LIN {X 0,Y 574.364,Z 450.837,A -85,B 0,C 180,E1 -2266.254,E2 -2266.254} C_VEL
LIN {X 0,Y 574.549,Z 436.626,A -85,B 0,C 180,E1 -2266.797,E2 -2266.797} C_VEL
LIN {X 0,Y 574.69,Z 422.126,A -85,B 0,C 180,E1 -2267.209,E2 -2267.209} C_VEL
LIN {X 0,Y 574.753,Z 406.706,A -85,B 0,C 180,E1 -2267.502,E2 -2267.502} C_VEL
LIN {X 0,Y 575.14,Z 251.823,A -85,B 0,C 180,E1 -2269.493,E2 -2269.493} C_VEL
LIN {X 0,Y 574.003,Z 245.811,A -85,B 0,C 180,E1 -2269.623,E2 -2269.623} C_VEL
LIN {X 0,Y 574.349,Z 220.396,A -85,B 0,C 180,E1 -2272.671,E2 -2272.671} C_VEL
LIN {X 0,Y 574.581,Z 198.331,A -85,B 0,C 180,E1 -2275.347,E2 -2275.347} C_VEL
LIN {X 0,Y 574.295,Z 195.164,A -85,B 0,C 180,E1 -2275.749,E2 -2275.749} C_VEL
LIN {X 0,Y 573.262,Z 190.706,A -85,B 0,C 180,E1 -2276.38,E2 -2276.38} C_VEL
LIN {X 0,Y 573.262,Z 190.698,A -85,B 0,C 180,E1 -2279.365,E2 -2279.365} C_VEL
LIN {X 0,Y 573.247,Z 190.706,A -85,B 0,C 180,E1 -2282.227,E2 -2282.227} C_VEL
LIN {X 0,Y 573.235,Z 190.701,A -85,B 0,C 180,E1 -2284.771,E2 -2284.771} C_VEL
LIN {X 0,Y 573.249,Z 190.698,A -85,B 0,C 180,E1 -2287.165,E2 -2287.165} C_VEL
LIN {X 0,Y 573.243,Z 190.702,A -85,B 0,C 180,E1 -2289.606,E2 -2289.606} C_VEL
LIN {X 0,Y 573.237,Z 190.701,A -85,B 0,C 180,E1 -2292.641,E2 -2292.641} C_VEL
LIN {X 0,Y 573.229,Z 190.705,A -85,B 0,C 180,E1 -2295.666,E2 -2295.666} C_VEL
LIN {X 0,Y 573.239,Z 190.7,A -85,B 0,C 180,E1 -2298.544,E2 -2298.544} C_VEL
LIN {X 0,Y 573.243,Z 190.7,A -85,B 0,C 180,E1 -2301.299,E2 -2301.299} C_VEL
LIN {X 0,Y 573.257,Z 190.704,A -85,B 0,C 180,E1 -2304.011,E2 -2304.011} C_VEL
LIN {X 0,Y 573.277,Z 190.695,A -85,B 0,C 180,E1 -2306.518,E2 -2306.518} C_VEL
LIN {X 0,Y 573.236,Z 190.7,A -85,B 0,C 180,E1 -2309.115,E2 -2309.115} C_VEL
LIN {X 0,Y 573.256,Z 190.703,A -85,B 0,C 180,E1 -2311.968,E2 -2311.968} C_VEL
LIN {X 0,Y 573.245,Z 190.699,A -85,B 0,C 180,E1 -2314.59,E2 -2314.59} C_VEL
LIN {X 0,Y 573.231,Z 190.707,A -85,B 0,C 180,E1 -2317.662,E2 -2317.662} C_VEL
LIN {X 0,Y 573.248,Z 190.703,A -85,B 0,C 180,E1 -2319.923,E2 -2319.923} C_VEL
LIN {X 0,Y 573.254,Z 190.699,A -85,B 0,C 180,E1 -2322.988,E2 -2322.988} C_VEL
LIN {X 0,Y 573.264,Z 190.702,A -85,B 0,C 180,E1 -2325.807,E2 -2325.807} C_VEL
LIN {X 0,Y 573.273,Z 190.695,A -85,B 0,C 180,E1 -2328.734,E2 -2328.734} C_VEL
LIN {X 0,Y 573.298,Z 190.701,A -85,B 0,C 180,E1 -2331.541,E2 -2331.541} C_VEL
LIN {X 0,Y 573.285,Z 190.693,A -85,B 0,C 180,E1 -2334.372,E2 -2334.372} C_VEL
LIN {X 0,Y 573.298,Z 190.695,A -85,B 0,C 180,E1 -2337.892,E2 -2337.892} C_VEL
LIN {X 0,Y 573.329,Z 190.688,A -85,B 0,C 180,E1 -2340.702,E2 -2340.702} C_VEL
LIN {X 0,Y 573.233,Z 190.706,A -85,B 0,C 180,E1 -2343.515,E2 -2343.515} C_VEL
LIN {X 0,Y 573.287,Z 190.698,A -85,B 0,C 180,E1 -2345.628,E2 -2345.628} C_VEL
LIN {X 0,Y 573.299,Z 190.691,A -85,B 0,C 180,E1 -2348.459,E2 -2348.459} C_VEL
LIN {X 0,Y 573.29,Z 190.701,A -85,B 0,C 180,E1 -2351.312,E2 -2351.312} C_VEL
LIN {X 0,Y 573.272,Z 190.696,A -85,B 0,C 180,E1 -2354.425,E2 -2354.425} C_VEL
LIN {X 0,Y 573.251,Z 190.707,A -85,B 0,C 180,E1 -2357.112,E2 -2357.112} C_VEL
LIN {X 0,Y 573.246,Z 190.698,A -85,B 0,C 180,E1 -2360.077,E2 -2360.077} C_VEL
LIN {X 0,Y 573.225,Z 190.71,A -85,B 0,C 180,E1 -2363.1,E2 -2363.1} C_VEL
LIN {X 0,Y 573.243,Z 190.699,A -85,B 0,C 180,E1 -2364.399,E2 -2364.399} C_VEL
LIN {X 0,Y 572.617,Z 190.785,A -85,B 0,C 180,E1 -2364.985,E2 -2364.985} C_VEL
LIN {X 0,Y 569.775,Z 191.14,A -85,B 0,C 180,E1 -2365.937,E2 -2365.937} C_VEL
LIN {X 0,Y 567.345,Z 191.442,A -85,B 0,C 180,E1 -2366.702,E2 -2366.702} C_VEL
LIN {X 0,Y 566.294,Z 191.569,A -85,B 0,C 180,E1 -2367.294,E2 -2367.294} C_VEL
LIN {X 0,Y 566.206,Z 191.578,A -85,B 0,C 180,E1 -2367.494,E2 -2367.494} C_VEL
LIN {X 0,Y 566.219,Z 191.574,A -85,B 0,C 180,E1 -2369.768,E2 -2369.768} C_VEL
LIN {X 0,Y 566.2,Z 191.579,A -85,B 0,C 180,E1 -2372.431,E2 -2372.431} C_VEL
LIN {X 0,Y 566.208,Z 191.584,A -85,B 0,C 180,E1 -2374.995,E2 -2374.995} C_VEL
LIN {X 0,Y 566.191,Z 191.579,A -85,B 0,C 180,E1 -2377.461,E2 -2377.461} C_VEL
LIN {X 0,Y 566.222,Z 191.574,A -85,B 0,C 180,E1 -2380.198,E2 -2380.198} C_VEL
LIN {X 0,Y 566.196,Z 191.582,A -85,B 0,C 180,E1 -2383.055,E2 -2383.055} C_VEL
LIN {X 0,Y 566.198,Z 191.577,A -85,B 0,C 180,E1 -2386.049,E2 -2386.049} C_VEL
LIN {X 0,Y 566.207,Z 191.584,A -85,B 0,C 180,E1 -2388.864,E2 -2388.864} C_VEL
LIN {X 0,Y 566.184,Z 191.578,A -85,B 0,C 180,E1 -2391.638,E2 -2391.638} C_VEL
LIN {X 0,Y 566.16,Z 191.586,A -85,B 0,C 180,E1 -2394.309,E2 -2394.309} C_VEL
LIN {X 0,Y 566.228,Z 191.579,A -85,B 0,C 180,E1 -2396.899,E2 -2396.899} C_VEL
LIN {X 0,Y 566.182,Z 191.58,A -85,B 0,C 180,E1 -2399.408,E2 -2399.408} C_VEL
LIN {X 0,Y 566.211,Z 191.578,A -85,B 0,C 180,E1 -2401.858,E2 -2401.858} C_VEL
LIN {X 0,Y 566.214,Z 191.582,A -85,B 0,C 180,E1 -2404.252,E2 -2404.252} C_VEL
LIN {X 0,Y 566.209,Z 191.685,A -85,B 0,C 180,E1 -2406.549,E2 -2406.549} C_VEL
LIN {X 0,Y 567.22,Z 197.326,A -85,B 0,C 180,E1 -2407.413,E2 -2407.413} C_VEL
LIN {X 0,Y 566.915,Z 216.903,A -85,B 0,C 180,E1 -2410.188,E2 -2410.188} C_VEL
LIN {X 0,Y 568.489,Z 225.078,A -85,B 0,C 180,E1 -2410.358,E2 -2410.358} C_VEL
LIN {X 0,Y 567.967,Z 382.291,A -85,B 0,C 180,E1 -2412.415,E2 -2412.415} C_VEL
LIN {X 0,Y 567.819,Z 397.78,A -85,B 0,C 180,E1 -2412.766,E2 -2412.766} C_VEL
LIN {X 0,Y 567.62,Z 413.086,A -85,B 0,C 180,E1 -2413.27,E2 -2413.27} C_VEL
LIN {X 0,Y 567.399,Z 427.739,A -85,B 0,C 180,E1 -2413.911,E2 -2413.911} C_VEL
LIN {X 0,Y 567.156,Z 441.053,A -85,B 0,C 180,E1 -2414.641,E2 -2414.641} C_VEL
LIN {X 0,Y 566.917,Z 453.985,A -85,B 0,C 180,E1 -2415.508,E2 -2415.508} C_VEL
LIN {X 0,Y 566.653,Z 466.893,A -85,B 0,C 180,E1 -2416.553,E2 -2416.553} C_VEL
LIN {X 0,Y 566.462,Z 478.088,A -85,B 0,C 180,E1 -2417.642,E2 -2417.642} C_VEL
LIN {X 0,Y 566.263,Z 488.18,A -85,B 0,C 180,E1 -2418.81,E2 -2418.81} C_VEL
LIN {X 0,Y 566.133,Z 498.005,A -85,B 0,C 180,E1 -2420.172,E2 -2420.172} C_VEL
LIN {X 0,Y 566.063,Z 505.495,A -85,B 0,C 180,E1 -2421.432,E2 -2421.432} C_VEL
LIN {X 0,Y 565.975,Z 512.5,A -85,B 0,C 180,E1 -2422.867,E2 -2422.867} C_VEL
LIN {X 0,Y 565.982,Z 518.009,A -85,B 0,C 180,E1 -2424.299,E2 -2424.299} C_VEL
LIN {X 0,Y 565.913,Z 522.178,A -85,B 0,C 180,E1 -2425.727,E2 -2425.727} C_VEL
LIN {X 0,Y 565.872,Z 525.113,A -85,B 0,C 180,E1 -2427.152,E2 -2427.152} C_VEL
LIN {X 0,Y 565.842,Z 526.879,A -85,B 0,C 180,E1 -2428.577,E2 -2428.577} C_VEL
LIN {X 0,Y 565.837,Z 527.496,A -85,B 0,C 180,E1 -2430,E2 -2430} C_VEL
LIN {X 0,Y 565.844,Z 526.941,A -85,B 0,C 180,E1 -2431.423,E2 -2431.423} C_VEL
LIN {X 0,Y 565.874,Z 525.257,A -85,B 0,C 180,E1 -2432.847,E2 -2432.847} C_VEL
LIN {X 0,Y 565.913,Z 522.404,A -85,B 0,C 180,E1 -2434.273,E2 -2434.273} C_VEL
LIN {X 0,Y 565.975,Z 518.318,A -85,B 0,C 180,E1 -2435.701,E2 -2435.701} C_VEL
LIN {X 0,Y 565.975,Z 512.904,A -85,B 0,C 180,E1 -2437.133,E2 -2437.133} C_VEL
LIN {X 0,Y 566.061,Z 506.004,A -85,B 0,C 180,E1 -2438.568,E2 -2438.568} C_VEL
LIN {X 0,Y 566.177,Z 497.395,A -85,B 0,C 180,E1 -2440.008,E2 -2440.008} C_VEL
LIN {X 0,Y 566.25,Z 488.954,A -85,B 0,C 180,E1 -2441.183,E2 -2441.183} C_VEL
LIN {X 0,Y 566.436,Z 478.917,A -85,B 0,C 180,E1 -2442.358,E2 -2442.358} C_VEL
LIN {X 0,Y 566.668,Z 466.874,A -85,B 0,C 180,E1 -2443.538,E2 -2443.538} C_VEL
LIN {X 0,Y 566.878,Z 455.249,A -85,B 0,C 180,E1 -2444.488,E2 -2444.488} C_VEL
LIN {X 0,Y 567.091,Z 442.476,A -85,B 0,C 180,E1 -2445.361,E2 -2445.361} C_VEL
LIN {X 0,Y 567.376,Z 429.466,A -85,B 0,C 180,E1 -2446.09,E2 -2446.09} C_VEL
LIN {X 0,Y 567.567,Z 415.275,A -85,B 0,C 180,E1 -2446.732,E2 -2446.732} C_VEL
LIN {X 0,Y 567.789,Z 400.729,A -85,B 0,C 180,E1 -2447.235,E2 -2447.235} C_VEL
LIN {X 0,Y 567.928,Z 385.332,A -85,B 0,C 180,E1 -2447.615,E2 -2447.615} C_VEL
LIN {X 0,Y 568.048,Z 363.9,A -85,B 0,C 180,E1 -2447.932,E2 -2447.932} C_VEL
LIN {X 0,Y 568.437,Z 224.034,A -85,B 0,C 180,E1 -2449.748,E2 -2449.748} C_VEL
LIN {X 0,Y 566.883,Z 216.905,A -85,B 0,C 180,E1 -2449.903,E2 -2449.903} C_VEL
LIN {X 0,Y 567.213,Z 199.31,A -85,B 0,C 180,E1 -2452.395,E2 -2452.395} C_VEL
LIN {X 0,Y 567.005,Z 195.381,A -85,B 0,C 180,E1 -2452.971,E2 -2452.971} C_VEL
LIN {X 0,Y 566.191,Z 191.587,A -85,B 0,C 180,E1 -2453.573,E2 -2453.573} C_VEL
LIN {X 0,Y 566.215,Z 191.583,A -85,B 0,C 180,E1 -2455.748,E2 -2455.748} C_VEL
LIN {X 0,Y 566.202,Z 191.579,A -85,B 0,C 180,E1 -2458.201,E2 -2458.201} C_VEL
LIN {X 0,Y 566.192,Z 191.582,A -85,B 0,C 180,E1 -2461.076,E2 -2461.076} C_VEL
LIN {X 0,Y 566.21,Z 191.581,A -85,B 0,C 180,E1 -2463.734,E2 -2463.734} C_VEL
LIN {X 0,Y 566.205,Z 191.576,A -85,B 0,C 180,E1 -2466.569,E2 -2466.569} C_VEL
LIN {X 0,Y 566.208,Z 191.58,A -85,B 0,C 180,E1 -2469.685,E2 -2469.685} C_VEL
LIN {X 0,Y 566.21,Z 191.576,A -85,B 0,C 180,E1 -2472.086,E2 -2472.086} C_VEL
LIN {X 0,Y 566.169,Z 191.586,A -85,B 0,C 180,E1 -2475.035,E2 -2475.035} C_VEL
LIN {X 0,Y 566.212,Z 191.573,A -85,B 0,C 180,E1 -2478.135,E2 -2478.135} C_VEL
LIN {X 0,Y 566.217,Z 191.577,A -85,B 0,C 180,E1 -2480.726,E2 -2480.726} C_VEL
LIN {X 0,Y 566.212,Z 191.576,A -85,B 0,C 180,E1 -2483.783,E2 -2483.783} C_VEL
LIN {X 0,Y 566.205,Z 191.576,A -85,B 0,C 180,E1 -2486.265,E2 -2486.265} C_VEL
LIN {X 0,Y 566.196,Z 191.58,A -85,B 0,C 180,E1 -2488.921,E2 -2488.921} C_VEL
LIN {X 0,Y 566.189,Z 191.586,A -85,B 0,C 180,E1 -2491.046,E2 -2491.046} C_VEL
LIN {X 0,Y 566.208,Z 191.578,A -85,B 0,C 180,E1 -2493.458,E2 -2493.458} C_VEL
LIN {X 0,Y 566.192,Z 191.578,A -85,B 0,C 180,E1 -2495.819,E2 -2495.819} C_VEL
LIN {X 0,Y 566.208,Z 191.584,A -85,B 0,C 180,E1 -2498.902,E2 -2498.902} C_VEL
LIN {X 0,Y 566.204,Z 191.581,A -85,B 0,C 180,E1 -2501.172,E2 -2501.172} C_VEL
LIN {X 0,Y 566.213,Z 191.577,A -85,B 0,C 180,E1 -2503.412,E2 -2503.412} C_VEL
LIN {X 0,Y 566.193,Z 191.578,A -85,B 0,C 180,E1 -2506.359,E2 -2506.359} C_VEL
LIN {X 0,Y 566.266,Z 191.575,A -85,B 0,C 180,E1 -2508.654,E2 -2508.654} C_VEL
LIN {X 0,Y 566.226,Z 191.574,A -85,B 0,C 180,E1 -2511.434,E2 -2511.434} C_VEL
LIN {X 0,Y 566.254,Z 191.572,A -85,B 0,C 180,E1 -2514.302,E2 -2514.302} C_VEL
LIN {X 0,Y 566.269,Z 191.568,A -85,B 0,C 180,E1 -2517.866,E2 -2517.866} C_VEL
LIN {X 0,Y 566.3,Z 191.573,A -85,B 0,C 180,E1 -2520.711,E2 -2520.711} C_VEL
LIN {X 0,Y 566.271,Z 191.573,A -85,B 0,C 180,E1 -2522.845,E2 -2522.845} C_VEL
LIN {X 0,Y 566.252,Z 191.57,A -85,B 0,C 180,E1 -2525.698,E2 -2525.698} C_VEL
LIN {X 0,Y 566.239,Z 191.58,A -85,B 0,C 180,E1 -2528.565,E2 -2528.565} C_VEL
LIN {X 0,Y 566.241,Z 191.571,A -85,B 0,C 180,E1 -2531.454,E2 -2531.454} C_VEL
LIN {X 0,Y 566.224,Z 191.583,A -85,B 0,C 180,E1 -2534.507,E2 -2534.507} C_VEL
LIN {X 0,Y 566.195,Z 191.576,A -85,B 0,C 180,E1 -2537.332,E2 -2537.332} C_VEL
LIN {X 0,Y 566.211,Z 191.585,A -85,B 0,C 180,E1 -2540.337,E2 -2540.337} C_VEL
LIN {X 0,Y 566.181,Z 191.579,A -85,B 0,C 180,E1 -2543.404,E2 -2543.404} C_VEL
LIN {X 0,Y 566.205,Z 191.577,A -85,B 0,C 180,E1 -2545.749,E2 -2545.749} C_VEL
LIN {X 0,Y 566.198,Z 191.586,A -85,B 0,C 180,E1 -2548.204,E2 -2548.204} C_VEL
LIN {X 0,Y 566.186,Z 191.582,A -85,B 0,C 180,E1 -2550.592,E2 -2550.592} C_VEL
LIN {X 0,Y 566.221,Z 191.573,A -85,B 0,C 180,E1 -2553.102,E2 -2553.102} C_VEL
LIN {X 0,Y 566.205,Z 191.579,A -85,B 0,C 180,E1 -2555.689,E2 -2555.689} C_VEL
LIN {X 0,Y 566.206,Z 191.578,A -85,B 0,C 180,E1 -2558.559,E2 -2558.559} C_VEL
LIN {X 0,Y 566.205,Z 191.573,A -85,B 0,C 180,E1 -2561.137,E2 -2561.137} C_VEL
LIN {X 0,Y 566.191,Z 191.587,A -85,B 0,C 180,E1 -2564.036,E2 -2564.036} C_VEL
LIN {X 0,Y 566.199,Z 191.577,A -85,B 0,C 180,E1 -2567.083,E2 -2567.083} C_VEL
LIN {X 0,Y 566.222,Z 191.581,A -85,B 0,C 180,E1 -2569.803,E2 -2569.803} C_VEL
LIN {X 0,Y 566.195,Z 191.577,A -85,B 0,C 180,E1 -2572.6,E2 -2572.6} C_VEL
LIN {X 0,Y 566.204,Z 191.577,A -85,B 0,C 180,E1 -2575.183,E2 -2575.183} C_VEL
LIN {X 0,Y 566.227,Z 191.582,A -85,B 0,C 180,E1 -2577.744,E2 -2577.744} C_VEL
LIN {X 0,Y 566.201,Z 191.581,A -85,B 0,C 180,E1 -2580.329,E2 -2580.329} C_VEL
LIN {X 0,Y 566.211,Z 191.584,A -85,B 0,C 180,E1 -2583.417,E2 -2583.417} C_VEL
LIN {X 0,Y 567.68,Z 198.141,A -85,B 0,C 180,E1 -2584.323,E2 -2584.323} C_VEL
LIN {X 0,Y 567.546,Z 214.98,A -85,B 0,C 180,E1 -2586.398,E2 -2586.398} C_VEL
LIN {X 0,Y 567.215,Z 237.563,A -85,B 0,C 180,E1 -2589.132,E2 -2589.132} C_VEL
LIN {X 0,Y 567.116,Z 245.947,A -85,B 0,C 180,E1 -2590.143,E2 -2590.143} C_VEL
LIN {X 0,Y 568.502,Z 254.36,A -85,B 0,C 180,E1 -2590.304,E2 -2590.304} C_VEL
LIN {X 0,Y 567.984,Z 411.957,A -85,B 0,C 180,E1 -2592.364,E2 -2592.364} C_VEL
LIN {X 0,Y 567.833,Z 427.718,A -85,B 0,C 180,E1 -2592.72,E2 -2592.72} C_VEL
LIN {X 0,Y 567.616,Z 443.047,A -85,B 0,C 180,E1 -2593.223,E2 -2593.223} C_VEL
LIN {X 0,Y 567.404,Z 456.784,A -85,B 0,C 180,E1 -2593.818,E2 -2593.818} C_VEL
LIN {X 0,Y 567.148,Z 470.255,A -85,B 0,C 180,E1 -2594.549,E2 -2594.549} C_VEL
LIN {X 0,Y 566.931,Z 482.527,A -85,B 0,C 180,E1 -2595.359,E2 -2595.359} C_VEL
LIN {X 0,Y 566.672,Z 495.296,A -85,B 0,C 180,E1 -2596.371,E2 -2596.371} C_VEL
LIN {X 0,Y 566.491,Z 506.752,A -85,B 0,C 180,E1 -2597.461,E2 -2597.461} C_VEL
LIN {X 0,Y 566.268,Z 517.313,A -85,B 0,C 180,E1 -2598.659,E2 -2598.659} C_VEL
LIN {X 0,Y 566.208,Z 525.858,A -85,B 0,C 180,E1 -2599.812,E2 -2599.812} C_VEL
LIN {X 0,Y 566.057,Z 533.736,A -85,B 0,C 180,E1 -2601.072,E2 -2601.072} C_VEL
LIN {X 0,Y 565.997,Z 541.091,A -85,B 0,C 180,E1 -2602.509,E2 -2602.509} C_VEL
LIN {X 0,Y 565.959,Z 546.923,A -85,B 0,C 180,E1 -2603.941,E2 -2603.941} C_VEL
LIN {X 0,Y 565.866,Z 550.386,A -85,B 0,C 180,E1 -2605.013,E2 -2605.013} C_VEL
LIN {X 0,Y 565.909,Z 553.889,A -85,B 0,C 180,E1 -2606.44,E2 -2606.44} C_VEL
LIN {X 0,Y 565.839,Z 556.191,A -85,B 0,C 180,E1 -2607.865,E2 -2607.865} C_VEL
LIN {X 0,Y 565.839,Z 557.349,A -85,B 0,C 180,E1 -2609.288,E2 -2609.288} C_VEL
LIN {X 0,Y 565.839,Z 557.348,A -85,B 0,C 180,E1 -2610.712,E2 -2610.712} C_VEL
LIN {X 0,Y 565.839,Z 556.189,A -85,B 0,C 180,E1 -2612.135,E2 -2612.135} C_VEL
LIN {X 0,Y 565.909,Z 553.886,A -85,B 0,C 180,E1 -2613.56,E2 -2613.56} C_VEL
LIN {X 0,Y 565.866,Z 550.386,A -85,B 0,C 180,E1 -2614.987,E2 -2614.987} C_VEL
LIN {X 0,Y 565.942,Z 545.609,A -85,B 0,C 180,E1 -2616.417,E2 -2616.417} C_VEL
LIN {X 0,Y 566.014,Z 539.423,A -85,B 0,C 180,E1 -2617.85,E2 -2617.85} C_VEL
LIN {X 0,Y 566.071,Z 531.648,A -85,B 0,C 180,E1 -2619.288,E2 -2619.288} C_VEL
LIN {X 0,Y 566.239,Z 523.37,A -85,B 0,C 180,E1 -2620.549,E2 -2620.549} C_VEL
LIN {X 0,Y 566.367,Z 513.394,A -85,B 0,C 180,E1 -2621.814,E2 -2621.814} C_VEL
LIN {X 0,Y 566.585,Z 503.19,A -85,B 0,C 180,E1 -2622.901,E2 -2622.901} C_VEL
LIN {X 0,Y 566.799,Z 491.023,A -85,B 0,C 180,E1 -2623.992,E2 -2623.992} C_VEL
LIN {X 0,Y 567.039,Z 478.343,A -85,B 0,C 180,E1 -2624.936,E2 -2624.936} C_VEL
LIN {X 0,Y 567.278,Z 465.516,A -85,B 0,C 180,E1 -2625.724,E2 -2625.724} C_VEL
LIN {X 0,Y 567.498,Z 450.834,A -85,B 0,C 180,E1 -2626.456,E2 -2626.456} C_VEL
LIN {X 0,Y 567.72,Z 436.625,A -85,B 0,C 180,E1 -2627.005,E2 -2627.005} C_VEL
LIN {X 0,Y 567.922,Z 422.257,A -85,B 0,C 180,E1 -2627.417,E2 -2627.417} C_VEL
LIN {X 0,Y 567.982,Z 407.822,A -85,B 0,C 180,E1 -2627.7,E2 -2627.7} C_VEL
LIN {X 0,Y 568.494,Z 253.496,A -85,B 0,C 180,E1 -2629.708,E2 -2629.708} C_VEL
LIN {X 0,Y 567.136,Z 245.837,A -85,B 0,C 180,E1 -2629.867,E2 -2629.867} C_VEL
LIN {X 0,Y 567.466,Z 221.81,A -85,B 0,C 180,E1 -2632.769,E2 -2632.769} C_VEL
LIN {X 0,Y 567.755,Z 199.933,A -85,B 0,C 180,E1 -2635.452,E2 -2635.452} C_VEL
LIN {X 0,Y 567.38,Z 196.566,A -85,B 0,C 180,E1 -2635.889,E2 -2635.889} C_VEL
LIN {X 0,Y 566.211,Z 191.584,A -85,B 0,C 180,E1 -2636.583,E2 -2636.583} C_VEL
LIN {X 0,Y 566.201,Z 191.58,A -85,B 0,C 180,E1 -2639.671,E2 -2639.671} C_VEL
LIN {X 0,Y 566.2,Z 191.58,A -85,B 0,C 180,E1 -2642.429,E2 -2642.429} C_VEL
LIN {X 0,Y 566.196,Z 191.576,A -85,B 0,C 180,E1 -2644.992,E2 -2644.992} C_VEL
LIN {X 0,Y 566.193,Z 191.579,A -85,B 0,C 180,E1 -2647.46,E2 -2647.46} C_VEL
LIN {X 0,Y 566.222,Z 191.581,A -85,B 0,C 180,E1 -2650.197,E2 -2650.197} C_VEL
LIN {X 0,Y 566.199,Z 191.576,A -85,B 0,C 180,E1 -2653.053,E2 -2653.053} C_VEL
LIN {X 0,Y 566.192,Z 191.585,A -85,B 0,C 180,E1 -2656.048,E2 -2656.048} C_VEL
LIN {X 0,Y 566.206,Z 191.575,A -85,B 0,C 180,E1 -2658.863,E2 -2658.863} C_VEL
LIN {X 0,Y 566.184,Z 191.583,A -85,B 0,C 180,E1 -2661.637,E2 -2661.637} C_VEL
LIN {X 0,Y 566.205,Z 191.578,A -85,B 0,C 180,E1 -2664.311,E2 -2664.311} C_VEL
LIN {X 0,Y 566.221,Z 191.572,A -85,B 0,C 180,E1 -2666.898,E2 -2666.898} C_VEL
LIN {X 0,Y 566.186,Z 191.581,A -85,B 0,C 180,E1 -2669.408,E2 -2669.408} C_VEL
LIN {X 0,Y 566.22,Z 191.582,A -85,B 0,C 180,E1 -2671.858,E2 -2671.858} C_VEL
LIN {X 0,Y 566.205,Z 191.578,A -85,B 0,C 180,E1 -2674.251,E2 -2674.251} C_VEL
LIN {X 0,Y 566.183,Z 191.577,A -85,B 0,C 180,E1 -2676.713,E2 -2676.713} C_VEL
LIN {X 0,Y 566.211,Z 191.582,A -85,B 0,C 180,E1 -2679.663,E2 -2679.663} C_VEL
LIN {X 0,Y 566.195,Z 191.577,A -85,B 0,C 180,E1 -2682.668,E2 -2682.668} C_VEL
LIN {X 0,Y 566.224,Z 191.582,A -85,B 0,C 180,E1 -2685.627,E2 -2685.627} C_VEL
LIN {X 0,Y 566.265,Z 191.568,A -85,B 0,C 180,E1 -2688.654,E2 -2688.654} C_VEL
LIN {X 0,Y 566.239,Z 191.58,A -85,B 0,C 180,E1 -2691.435,E2 -2691.435} C_VEL
LIN {X 0,Y 566.252,Z 191.57,A -85,B 0,C 180,E1 -2694.302,E2 -2694.302} C_VEL
LIN {X 0,Y 566.27,Z 191.571,A -85,B 0,C 180,E1 -2697.866,E2 -2697.866} C_VEL
LIN {X 0,Y 566.298,Z 191.564,A -85,B 0,C 180,E1 -2700.711,E2 -2700.711} C_VEL
LIN {X 0,Y 566.27,Z 191.57,A -85,B 0,C 180,E1 -2702.846,E2 -2702.846} C_VEL
LIN {X 0,Y 566.254,Z 191.573,A -85,B 0,C 180,E1 -2705.698,E2 -2705.698} C_VEL
LIN {X 0,Y 566.24,Z 191.571,A -85,B 0,C 180,E1 -2708.566,E2 -2708.566} C_VEL
LIN {X 0,Y 566.242,Z 191.577,A -85,B 0,C 180,E1 -2711.454,E2 -2711.454} C_VEL
LIN {X 0,Y 566.225,Z 191.574,A -85,B 0,C 180,E1 -2714.507,E2 -2714.507} C_VEL
LIN {X 0,Y 566.195,Z 191.584,A -85,B 0,C 180,E1 -2717.332,E2 -2717.332} C_VEL
LIN {X 0,Y 566.206,Z 191.575,A -85,B 0,C 180,E1 -2720.338,E2 -2720.338} C_VEL
LIN {X 0,Y 566.181,Z 191.582,A -85,B 0,C 180,E1 -2723.404,E2 -2723.404} C_VEL
LIN {X 0,Y 566.207,Z 191.571,A -85,B 0,C 180,E1 -2725.749,E2 -2725.749} C_VEL
LIN {X 0,Y 566.206,Z 191.578,A -85,B 0,C 180,E1 -2727.494,E2 -2727.494} C_VEL
LIN {X 0,Y 565.53,Z 191.661,A -85,B 0,C 180,E1 -2728.088,E2 -2728.088} C_VEL
LIN {X 0,Y 562.667,Z 192.025,A -85,B 0,C 180,E1 -2729.051,E2 -2729.051} C_VEL
LIN {X 0,Y 560.256,Z 192.321,A -85,B 0,C 180,E1 -2729.827,E2 -2729.827} C_VEL
LIN {X 0,Y 559.227,Z 192.447,A -85,B 0,C 180,E1 -2730.426,E2 -2730.426} C_VEL
LIN {X 0,Y 559.146,Z 192.458,A -85,B 0,C 180,E1 -2730.628,E2 -2730.628} C_VEL
LIN {X 0,Y 559.158,Z 192.454,A -85,B 0,C 180,E1 -2733.575,E2 -2733.575} C_VEL
LIN {X 0,Y 559.163,Z 192.456,A -85,B 0,C 180,E1 -2736.449,E2 -2736.449} C_VEL
LIN {X 0,Y 559.173,Z 192.459,A -85,B 0,C 180,E1 -2738.934,E2 -2738.934} C_VEL
LIN {X 0,Y 559.186,Z 192.449,A -85,B 0,C 180,E1 -2741.768,E2 -2741.768} C_VEL
LIN {X 0,Y 559.135,Z 192.465,A -85,B 0,C 180,E1 -2744.74,E2 -2744.74} C_VEL
LIN {X 0,Y 559.161,Z 192.456,A -85,B 0,C 180,E1 -2747.258,E2 -2747.258} C_VEL
LIN {X 0,Y 559.177,Z 192.454,A -85,B 0,C 180,E1 -2750.135,E2 -2750.135} C_VEL
LIN {X 0,Y 559.138,Z 192.462,A -85,B 0,C 180,E1 -2752.892,E2 -2752.892} C_VEL
LIN {X 0,Y 559.164,Z 192.456,A -85,B 0,C 180,E1 -2756.052,E2 -2756.052} C_VEL
LIN {X 0,Y 559.157,Z 192.459,A -85,B 0,C 180,E1 -2758.982,E2 -2758.982} C_VEL
LIN {X 0,Y 559.167,Z 192.454,A -85,B 0,C 180,E1 -2761.619,E2 -2761.619} C_VEL
LIN {X 0,Y 559.181,Z 192.455,A -85,B 0,C 180,E1 -2763.904,E2 -2763.904} C_VEL
LIN {X 0,Y 559.161,Z 192.485,A -85,B 0,C 180,E1 -2766.328,E2 -2766.328} C_VEL
LIN {X 0,Y 560.343,Z 198.825,A -85,B 0,C 180,E1 -2767.315,E2 -2767.315} C_VEL
LIN {X 0,Y 560.027,Z 217.038,A -85,B 0,C 180,E1 -2769.934,E2 -2769.934} C_VEL
LIN {X 0,Y 561.825,Z 225.981,A -85,B 0,C 180,E1 -2770.125,E2 -2770.125} C_VEL
LIN {X 0,Y 561.211,Z 382.553,A -85,B 0,C 180,E1 -2772.2,E2 -2772.2} C_VEL
LIN {X 0,Y 561.052,Z 397.801,A -85,B 0,C 180,E1 -2772.552,E2 -2772.552} C_VEL
LIN {X 0,Y 560.82,Z 413.099,A -85,B 0,C 180,E1 -2773.061,E2 -2773.061} C_VEL
LIN {X 0,Y 560.561,Z 427.747,A -85,B 0,C 180,E1 -2773.709,E2 -2773.709} C_VEL
LIN {X 0,Y 560.258,Z 441.064,A -85,B 0,C 180,E1 -2774.447,E2 -2774.447} C_VEL
LIN {X 0,Y 559.983,Z 454.396,A -85,B 0,C 180,E1 -2775.354,E2 -2775.354} C_VEL
LIN {X 0,Y 559.69,Z 466.9,A -85,B 0,C 180,E1 -2776.383,E2 -2776.383} C_VEL
LIN {X 0,Y 559.486,Z 478.093,A -85,B 0,C 180,E1 -2777.486,E2 -2777.486} C_VEL
LIN {X 0,Y 559.228,Z 488.789,A -85,B 0,C 180,E1 -2778.743,E2 -2778.743} C_VEL
LIN {X 0,Y 559.095,Z 498.008,A -85,B 0,C 180,E1 -2780.047,E2 -2780.047} C_VEL
LIN {X 0,Y 559.002,Z 505.498,A -85,B 0,C 180,E1 -2781.323,E2 -2781.323} C_VEL
LIN {X 0,Y 558.901,Z 512.502,A -85,B 0,C 180,E1 -2782.776,E2 -2782.776} C_VEL
LIN {X 0,Y 558.888,Z 518.011,A -85,B 0,C 180,E1 -2784.226,E2 -2784.226} C_VEL
LIN {X 0,Y 558.808,Z 522.178,A -85,B 0,C 180,E1 -2785.672,E2 -2785.672} C_VEL
LIN {X 0,Y 558.793,Z 525.112,A -85,B 0,C 180,E1 -2787.116,E2 -2787.116} C_VEL
LIN {X 0,Y 558.742,Z 526.879,A -85,B 0,C 180,E1 -2788.559,E2 -2788.559} C_VEL
LIN {X 0,Y 558.738,Z 527.496,A -85,B 0,C 180,E1 -2790,E2 -2790} C_VEL
LIN {X 0,Y 558.744,Z 526.94,A -85,B 0,C 180,E1 -2791.441,E2 -2791.441} C_VEL
LIN {X 0,Y 558.795,Z 525.256,A -85,B 0,C 180,E1 -2792.884,E2 -2792.884} C_VEL
LIN {X 0,Y 558.808,Z 522.403,A -85,B 0,C 180,E1 -2794.328,E2 -2794.328} C_VEL
LIN {X 0,Y 558.881,Z 518.317,A -85,B 0,C 180,E1 -2795.774,E2 -2795.774} C_VEL
LIN {X 0,Y 558.901,Z 512.901,A -85,B 0,C 180,E1 -2797.224,E2 -2797.224} C_VEL
LIN {X 0,Y 559.001,Z 506,A -85,B 0,C 180,E1 -2798.677,E2 -2798.677} C_VEL
LIN {X 0,Y 559.091,Z 498.573,A -85,B 0,C 180,E1 -2799.953,E2 -2799.953} C_VEL
LIN {X 0,Y 559.215,Z 489.513,A -85,B 0,C 180,E1 -2801.25,E2 -2801.25} C_VEL
LIN {X 0,Y 559.451,Z 478.911,A -85,B 0,C 180,E1 -2802.515,E2 -2802.515} C_VEL
LIN {X 0,Y 559.696,Z 466.867,A -85,B 0,C 180,E1 -2803.71,E2 -2803.71} C_VEL
LIN {X 0,Y 559.998,Z 454.177,A -85,B 0,C 180,E1 -2804.751,E2 -2804.751} C_VEL
LIN {X 0,Y 560.272,Z 441.013,A -85,B 0,C 180,E1 -2805.646,E2 -2805.646} C_VEL
LIN {X 0,Y 560.551,Z 427.686,A -85,B 0,C 180,E1 -2806.385,E2 -2806.385} C_VEL
LIN {X 0,Y 560.842,Z 412.997,A -85,B 0,C 180,E1 -2807.032,E2 -2807.032} C_VEL
LIN {X 0,Y 561.05,Z 398.351,A -85,B 0,C 180,E1 -2807.521,E2 -2807.521} C_VEL
LIN {X 0,Y 561.232,Z 382.449,A -85,B 0,C 180,E1 -2807.891,E2 -2807.891} C_VEL
LIN {X 0,Y 561.779,Z 225.243,A -85,B 0,C 180,E1 -2809.976,E2 -2809.976} C_VEL
LIN {X 0,Y 560.033,Z 216.928,A -85,B 0,C 180,E1 -2810.173,E2 -2810.173} C_VEL
LIN {X 0,Y 560.333,Z 198.134,A -85,B 0,C 180,E1 -2812.88,E2 -2812.88} C_VEL
LIN {X 0,Y 559.166,Z 192.462,A -85,B 0,C 180,E1 -2813.789,E2 -2813.789} C_VEL
LIN {X 0,Y 559.181,Z 192.456,A -85,B 0,C 180,E1 -2816.096,E2 -2816.096} C_VEL
LIN {X 0,Y 559.162,Z 192.455,A -85,B 0,C 180,E1 -2818.529,E2 -2818.529} C_VEL
LIN {X 0,Y 559.147,Z 192.462,A -85,B 0,C 180,E1 -2821.273,E2 -2821.273} C_VEL
LIN {X 0,Y 559.165,Z 192.456,A -85,B 0,C 180,E1 -2823.949,E2 -2823.949} C_VEL
LIN {X 0,Y 559.141,Z 192.461,A -85,B 0,C 180,E1 -2827.107,E2 -2827.107} C_VEL
LIN {X 0,Y 559.165,Z 192.454,A -85,B 0,C 180,E1 -2829.942,E2 -2829.942} C_VEL
LIN {X 0,Y 559.16,Z 192.455,A -85,B 0,C 180,E1 -2832.742,E2 -2832.742} C_VEL
LIN {X 0,Y 559.148,Z 192.457,A -85,B 0,C 180,E1 -2835.76,E2 -2835.76} C_VEL
LIN {X 0,Y 559.186,Z 192.449,A -85,B 0,C 180,E1 -2838.232,E2 -2838.232} C_VEL
LIN {X 0,Y 559.172,Z 192.46,A -85,B 0,C 180,E1 -2841.19,E2 -2841.19} C_VEL
LIN {X 0,Y 559.167,Z 192.453,A -85,B 0,C 180,E1 -2843.791,E2 -2843.791} C_VEL
LIN {X 0,Y 559.158,Z 192.454,A -85,B 0,C 180,E1 -2846.425,E2 -2846.425} C_VEL
LIN {X 0,Y 559.159,Z 192.457,A -85,B 0,C 180,E1 -2848.981,E2 -2848.981} C_VEL
LIN {X 0,Y 559.163,Z 192.455,A -85,B 0,C 180,E1 -2851.618,E2 -2851.618} C_VEL
LIN {X 0,Y 559.173,Z 192.451,A -85,B 0,C 180,E1 -2853.902,E2 -2853.902} C_VEL
LIN {X 0,Y 559.149,Z 192.458,A -85,B 0,C 180,E1 -2856.567,E2 -2856.567} C_VEL
LIN {X 0,Y 559.177,Z 192.454,A -85,B 0,C 180,E1 -2859.395,E2 -2859.395} C_VEL
LIN {X 0,Y 559.146,Z 192.454,A -85,B 0,C 180,E1 -2861.686,E2 -2861.686} C_VEL
LIN {X 0,Y 559.163,Z 192.453,A -85,B 0,C 180,E1 -2863.948,E2 -2863.948} C_VEL
LIN {X 0,Y 559.166,Z 192.452,A -85,B 0,C 180,E1 -2866.184,E2 -2866.184} C_VEL
LIN {X 0,Y 559.201,Z 192.452,A -85,B 0,C 180,E1 -2869.134,E2 -2869.134} C_VEL
LIN {X 0,Y 559.198,Z 192.449,A -85,B 0,C 180,E1 -2872.053,E2 -2872.053} C_VEL
LIN {X 0,Y 559.251,Z 192.447,A -85,B 0,C 180,E1 -2874.953,E2 -2874.953} C_VEL
LIN {X 0,Y 559.24,Z 192.443,A -85,B 0,C 180,E1 -2877.839,E2 -2877.839} C_VEL
LIN {X 0,Y 559.269,Z 192.449,A -85,B 0,C 180,E1 -2880.72,E2 -2880.72} C_VEL
LIN {X 0,Y 559.236,Z 192.448,A -85,B 0,C 180,E1 -2882.881,E2 -2882.881} C_VEL
LIN {X 0,Y 559.221,Z 192.446,A -85,B 0,C 180,E1 -2885.77,E2 -2885.77} C_VEL
LIN {X 0,Y 559.194,Z 192.456,A -85,B 0,C 180,E1 -2888.674,E2 -2888.674} C_VEL
LIN {X 0,Y 559.199,Z 192.449,A -85,B 0,C 180,E1 -2891.6,E2 -2891.6} C_VEL
LIN {X 0,Y 559.189,Z 192.458,A -85,B 0,C 180,E1 -2894.596,E2 -2894.596} C_VEL
LIN {X 0,Y 559.155,Z 192.453,A -85,B 0,C 180,E1 -2897.557,E2 -2897.557} C_VEL
LIN {X 0,Y 559.166,Z 192.455,A -85,B 0,C 180,E1 -2899.838,E2 -2899.838} C_VEL
LIN {X 0,Y 559.134,Z 192.462,A -85,B 0,C 180,E1 -2902.153,E2 -2902.153} C_VEL
LIN {X 0,Y 559.17,Z 192.451,A -85,B 0,C 180,E1 -2905.187,E2 -2905.187} C_VEL
LIN {X 0,Y 559.184,Z 192.453,A -85,B 0,C 180,E1 -2907.712,E2 -2907.712} C_VEL
LIN {X 0,Y 559.16,Z 192.463,A -85,B 0,C 180,E1 -2910.182,E2 -2910.182} C_VEL
LIN {X 0,Y 559.168,Z 192.454,A -85,B 0,C 180,E1 -2912.714,E2 -2912.714} C_VEL
LIN {X 0,Y 559.15,Z 192.455,A -85,B 0,C 180,E1 -2915.322,E2 -2915.322} C_VEL
LIN {X 0,Y 559.127,Z 192.465,A -85,B 0,C 180,E1 -2918.018,E2 -2918.018} C_VEL
LIN {X 0,Y 559.17,Z 192.45,A -85,B 0,C 180,E1 -2920.811,E2 -2920.811} C_VEL
LIN {X 0,Y 559.135,Z 192.462,A -85,B 0,C 180,E1 -2923.734,E2 -2923.734} C_VEL
LIN {X 0,Y 559.144,Z 192.456,A -85,B 0,C 180,E1 -2926.804,E2 -2926.804} C_VEL
LIN {X 0,Y 559.172,Z 192.452,A -85,B 0,C 180,E1 -2929.19,E2 -2929.19} C_VEL
LIN {X 0,Y 559.13,Z 192.464,A -85,B 0,C 180,E1 -2931.983,E2 -2931.983} C_VEL
LIN {X 0,Y 559.143,Z 192.456,A -85,B 0,C 180,E1 -2934.786,E2 -2934.786} C_VEL
LIN {X 0,Y 559.17,Z 192.456,A -85,B 0,C 180,E1 -2937.362,E2 -2937.362} C_VEL
LIN {X 0,Y 559.146,Z 192.462,A -85,B 0,C 180,E1 -2940.143,E2 -2940.143} C_VEL
LIN {X 0,Y 559.166,Z 192.459,A -85,B 0,C 180,E1 -2943.098,E2 -2943.098} C_VEL
LIN {X 0,Y 559.155,Z 192.466,A -85,B 0,C 180,E1 -2943.21,E2 -2943.21} C_VEL
LIN {X 0,Y 560.888,Z 200.214,A -85,B 0,C 180,E1 -2944.274,E2 -2944.274} C_VEL
LIN {X 0,Y 560.643,Z 220.046,A -85,B 0,C 180,E1 -2946.743,E2 -2946.743} C_VEL
LIN {X 0,Y 560.245,Z 245.283,A -85,B 0,C 180,E1 -2949.82,E2 -2949.82} C_VEL
LIN {X 0,Y 560.299,Z 246.175,A -85,B 0,C 180,E1 -2949.895,E2 -2949.895} C_VEL
LIN {X 0,Y 561.814,Z 255.082,A -85,B 0,C 180,E1 -2950.069,E2 -2950.069} C_VEL
LIN {X 0,Y 561.231,Z 412.039,A -85,B 0,C 180,E1 -2952.146,E2 -2952.146} C_VEL
LIN {X 0,Y 561.073,Z 427.243,A -85,B 0,C 180,E1 -2952.492,E2 -2952.492} C_VEL
LIN {X 0,Y 560.832,Z 441.81,A -85,B 0,C 180,E1 -2952.968,E2 -2952.968} C_VEL
LIN {X 0,Y 560.594,Z 454.808,A -85,B 0,C 180,E1 -2953.523,E2 -2953.523} C_VEL
LIN {X 0,Y 560.334,Z 468.681,A -85,B 0,C 180,E1 -2954.263,E2 -2954.263} C_VEL
LIN {X 0,Y 560.084,Z 480.936,A -85,B 0,C 180,E1 -2955.062,E2 -2955.062} C_VEL
LIN {X 0,Y 559.785,Z 493.158,A -85,B 0,C 180,E1 -2956.015,E2 -2956.015} C_VEL
LIN {X 0,Y 559.558,Z 504.97,A -85,B 0,C 180,E1 -2957.119,E2 -2957.119} C_VEL
LIN {X 0,Y 559.321,Z 514.906,A -85,B 0,C 180,E1 -2958.218,E2 -2958.218} C_VEL
LIN {X 0,Y 559.173,Z 524.624,A -85,B 0,C 180,E1 -2959.5,E2 -2959.5} C_VEL
LIN {X 0,Y 559.026,Z 532.725,A -85,B 0,C 180,E1 -2960.776,E2 -2960.776} C_VEL
LIN {X 0,Y 558.95,Z 539.425,A -85,B 0,C 180,E1 -2962.05,E2 -2962.05} C_VEL
LIN {X 0,Y 558.871,Z 545.607,A -85,B 0,C 180,E1 -2963.502,E2 -2963.502} C_VEL
LIN {X 0,Y 558.787,Z 550.387,A -85,B 0,C 180,E1 -2964.949,E2 -2964.949} C_VEL
LIN {X 0,Y 558.818,Z 553.889,A -85,B 0,C 180,E1 -2966.395,E2 -2966.395} C_VEL
LIN {X 0,Y 558.745,Z 556.191,A -85,B 0,C 180,E1 -2967.838,E2 -2967.838} C_VEL
LIN {X 0,Y 558.739,Z 557.348,A -85,B 0,C 180,E1 -2969.279,E2 -2969.279} C_VEL
LIN {X 0,Y 558.739,Z 557.348,A -85,B 0,C 180,E1 -2970.721,E2 -2970.721} C_VEL
LIN {X 0,Y 558.745,Z 556.188,A -85,B 0,C 180,E1 -2972.163,E2 -2972.163} C_VEL
LIN {X 0,Y 558.818,Z 553.885,A -85,B 0,C 180,E1 -2973.605,E2 -2973.605} C_VEL
LIN {X 0,Y 558.787,Z 550.387,A -85,B 0,C 180,E1 -2975.051,E2 -2975.051} C_VEL
LIN {X 0,Y 558.871,Z 545.609,A -85,B 0,C 180,E1 -2976.498,E2 -2976.498} C_VEL
LIN {X 0,Y 558.95,Z 539.422,A -85,B 0,C 180,E1 -2977.95,E2 -2977.95} C_VEL
LIN {X 0,Y 559.005,Z 531.646,A -85,B 0,C 180,E1 -2979.406,E2 -2979.406} C_VEL
LIN {X 0,Y 559.217,Z 523.369,A -85,B 0,C 180,E1 -2980.683,E2 -2980.683} C_VEL
LIN {X 0,Y 559.362,Z 513.394,A -85,B 0,C 180,E1 -2981.965,E2 -2981.965} C_VEL
LIN {X 0,Y 559.596,Z 503.189,A -85,B 0,C 180,E1 -2983.065,E2 -2983.065} C_VEL
LIN {X 0,Y 559.861,Z 491.023,A -85,B 0,C 180,E1 -2984.169,E2 -2984.169} C_VEL
LIN {X 0,Y 560.125,Z 478.69,A -85,B 0,C 180,E1 -2985.099,E2 -2985.099} C_VEL
LIN {X 0,Y 560.404,Z 465.513,A -85,B 0,C 180,E1 -2985.922,E2 -2985.922} C_VEL
LIN {X 0,Y 560.674,Z 450.831,A -85,B 0,C 180,E1 -2986.662,E2 -2986.662} C_VEL
LIN {X 0,Y 560.938,Z 436.625,A -85,B 0,C 180,E1 -2987.217,E2 -2987.217} C_VEL
LIN {X 0,Y 561.142,Z 422.165,A -85,B 0,C 180,E1 -2987.637,E2 -2987.637} C_VEL
LIN {X 0,Y 561.231,Z 407.668,A -85,B 0,C 180,E1 -2987.923,E2 -2987.923} C_VEL
LIN {X 0,Y 561.824,Z 254.784,A -85,B 0,C 180,E1 -2989.934,E2 -2989.934} C_VEL
LIN {X 0,Y 560.22,Z 245.839,A -85,B 0,C 180,E1 -2990.114,E2 -2990.114} C_VEL
LIN {X 0,Y 560.641,Z 220.045,A -85,B 0,C 180,E1 -2993.257,E2 -2993.257} C_VEL
LIN {X 0,Y 560.882,Z 200.256,A -85,B 0,C 180,E1 -2995.722,E2 -2995.722} C_VEL
LIN {X 0,Y 559.163,Z 192.46,A -85,B 0,C 180,E1 -2996.809,E2 -2996.809} C_VEL
LIN {X 0,Y 559.139,Z 192.458,A -85,B 0,C 180,E1 -2999.353,E2 -2999.353} C_VEL
LIN {X 0,Y 559.162,Z 192.458,A -85,B 0,C 180,E1 -3001.862,E2 -3001.862} C_VEL
LIN {X 0,Y 559.145,Z 192.459,A -85,B 0,C 180,E1 -3004.444,E2 -3004.444} C_VEL
LIN {X 0,Y 559.141,Z 192.456,A -85,B 0,C 180,E1 -3007.107,E2 -3007.107} C_VEL
LIN {X 0,Y 559.165,Z 192.461,A -85,B 0,C 180,E1 -3009.942,E2 -3009.942} C_VEL
LIN {X 0,Y 559.158,Z 192.454,A -85,B 0,C 180,E1 -3012.742,E2 -3012.742} C_VEL
LIN {X 0,Y 559.147,Z 192.461,A -85,B 0,C 180,E1 -3015.76,E2 -3015.76} C_VEL
LIN {X 0,Y 559.185,Z 192.455,A -85,B 0,C 180,E1 -3018.232,E2 -3018.232} C_VEL
LIN {X 0,Y 559.172,Z 192.452,A -85,B 0,C 180,E1 -3021.19,E2 -3021.19} C_VEL
LIN {X 0,Y 559.166,Z 192.461,A -85,B 0,C 180,E1 -3023.791,E2 -3023.791} C_VEL
LIN {X 0,Y 559.157,Z 192.454,A -85,B 0,C 180,E1 -3026.425,E2 -3026.425} C_VEL
LIN {X 0,Y 559.159,Z 192.453,A -85,B 0,C 180,E1 -3028.981,E2 -3028.981} C_VEL
LIN {X 0,Y 559.162,Z 192.46,A -85,B 0,C 180,E1 -3031.618,E2 -3031.618} C_VEL
LIN {X 0,Y 559.173,Z 192.459,A -85,B 0,C 180,E1 -3033.903,E2 -3033.903} C_VEL
LIN {X 0,Y 559.148,Z 192.453,A -85,B 0,C 180,E1 -3036.567,E2 -3036.567} C_VEL
LIN {X 0,Y 559.177,Z 192.452,A -85,B 0,C 180,E1 -3039.395,E2 -3039.395} C_VEL
LIN {X 0,Y 559.147,Z 192.464,A -85,B 0,C 180,E1 -3041.686,E2 -3041.686} C_VEL
LIN {X 0,Y 559.163,Z 192.457,A -85,B 0,C 180,E1 -3043.948,E2 -3043.948} C_VEL
LIN {X 0,Y 559.166,Z 192.454,A -85,B 0,C 180,E1 -3046.184,E2 -3046.184} C_VEL
LIN {X 0,Y 559.201,Z 192.452,A -85,B 0,C 180,E1 -3049.134,E2 -3049.134} C_VEL
LIN {X 0,Y 559.201,Z 192.45,A -85,B 0,C 180,E1 -3052.054,E2 -3052.054} C_VEL
LIN {X 0,Y 559.253,Z 192.444,A -85,B 0,C 180,E1 -3054.953,E2 -3054.953} C_VEL
LIN {X 0,Y 559.241,Z 192.446,A -85,B 0,C 180,E1 -3057.839,E2 -3057.839} C_VEL
LIN {X 0,Y 559.268,Z 192.44,A -85,B 0,C 180,E1 -3060.72,E2 -3060.72} C_VEL
LIN {X 0,Y 559.236,Z 192.447,A -85,B 0,C 180,E1 -3062.881,E2 -3062.881} C_VEL
LIN {X 0,Y 559.222,Z 192.448,A -85,B 0,C 180,E1 -3065.77,E2 -3065.77} C_VEL
LIN {X 0,Y 559.195,Z 192.449,A -85,B 0,C 180,E1 -3068.674,E2 -3068.674} C_VEL
LIN {X 0,Y 559.2,Z 192.451,A -85,B 0,C 180,E1 -3071.601,E2 -3071.601} C_VEL
LIN {X 0,Y 559.19,Z 192.451,A -85,B 0,C 180,E1 -3074.596,E2 -3074.596} C_VEL
LIN {X 0,Y 559.155,Z 192.457,A -85,B 0,C 180,E1 -3077.557,E2 -3077.557} C_VEL
LIN {X 0,Y 559.164,Z 192.453,A -85,B 0,C 180,E1 -3079.838,E2 -3079.838} C_VEL
LIN {X 0,Y 559.133,Z 192.457,A -85,B 0,C 180,E1 -3082.153,E2 -3082.153} C_VEL
LIN {X 0,Y 559.171,Z 192.454,A -85,B 0,C 180,E1 -3085.188,E2 -3085.188} C_VEL
LIN {X 0,Y 559.185,Z 192.45,A -85,B 0,C 180,E1 -3087.712,E2 -3087.712} C_VEL
LIN {X 0,Y 559.146,Z 192.458,A -85,B 0,C 180,E1 -3090.628,E2 -3090.628} C_VEL
LIN {X 0,Y 558.483,Z 192.546,A -85,B 0,C 180,E1 -3091.23,E2 -3091.23} C_VEL
LIN {X 0,Y 555.618,Z 192.901,A -85,B 0,C 180,E1 -3092.206,E2 -3092.206} C_VEL
LIN {X 0,Y 553.204,Z 193.203,A -85,B 0,C 180,E1 -3092.992,E2 -3092.992} C_VEL
LIN {X 0,Y 552.183,Z 193.323,A -85,B 0,C 180,E1 -3093.598,E2 -3093.598} C_VEL
LIN {X 0,Y 552.109,Z 193.331,A -85,B 0,C 180,E1 -3093.804,E2 -3093.804} C_VEL
LIN {X 0,Y 552.106,Z 193.339,A -85,B 0,C 180,E1 -3096.747,E2 -3096.747} C_VEL
LIN {X 0,Y 552.129,Z 193.329,A -85,B 0,C 180,E1 -3099.527,E2 -3099.527} C_VEL
LIN {X 0,Y 552.125,Z 193.332,A -85,B 0,C 180,E1 -3102.426,E2 -3102.426} C_VEL
LIN {X 0,Y 552.095,Z 193.334,A -85,B 0,C 180,E1 -3105.564,E2 -3105.564} C_VEL
LIN {X 0,Y 552.134,Z 193.337,A -85,B 0,C 180,E1 -3108.677,E2 -3108.677} C_VEL
LIN {X 0,Y 552.115,Z 193.332,A -85,B 0,C 180,E1 -3111.412,E2 -3111.412} C_VEL
LIN {X 0,Y 552.083,Z 193.338,A -85,B 0,C 180,E1 -3114.157,E2 -3114.157} C_VEL
LIN {X 0,Y 552.121,Z 193.338,A -85,B 0,C 180,E1 -3116.815,E2 -3116.815} C_VEL
LIN {X 0,Y 552.103,Z 193.334,A -85,B 0,C 180,E1 -3119.392,E2 -3119.392} C_VEL
LIN {X 0,Y 552.119,Z 193.334,A -85,B 0,C 180,E1 -3121.903,E2 -3121.903} C_VEL
LIN {X 0,Y 552.156,Z 193.335,A -85,B 0,C 180,E1 -3124.65,E2 -3124.65} C_VEL
LIN {X 0,Y 552.125,Z 193.447,A -85,B 0,C 180,E1 -3126.123,E2 -3126.123} C_VEL
LIN {X 0,Y 553.497,Z 200.347,A -85,B 0,C 180,E1 -3127.216,E2 -3127.216} C_VEL
LIN {X 0,Y 553.188,Z 217.492,A -85,B 0,C 180,E1 -3129.682,E2 -3129.682} C_VEL
LIN {X 0,Y 555.168,Z 226.93,A -85,B 0,C 180,E1 -3129.886,E2 -3129.886} C_VEL
LIN {X 0,Y 554.49,Z 382.283,A -85,B 0,C 180,E1 -3131.969,E2 -3131.969} C_VEL
LIN {X 0,Y 554.287,Z 397.916,A -85,B 0,C 180,E1 -3132.332,E2 -3132.332} C_VEL
LIN {X 0,Y 554.004,Z 413.174,A -85,B 0,C 180,E1 -3132.846,E2 -3132.846} C_VEL
LIN {X 0,Y 553.733,Z 427.772,A -85,B 0,C 180,E1 -3133.502,E2 -3133.502} C_VEL
LIN {X 0,Y 553.388,Z 441.075,A -85,B 0,C 180,E1 -3134.249,E2 -3134.249} C_VEL
LIN {X 0,Y 553.063,Z 454.733,A -85,B 0,C 180,E1 -3135.192,E2 -3135.192} C_VEL
LIN {X 0,Y 552.723,Z 466.907,A -85,B 0,C 180,E1 -3136.208,E2 -3136.208} C_VEL
LIN {X 0,Y 552.488,Z 478.099,A -85,B 0,C 180,E1 -3137.325,E2 -3137.325} C_VEL
LIN {X 0,Y 552.199,Z 489.343,A -85,B 0,C 180,E1 -3138.672,E2 -3138.672} C_VEL
LIN {X 0,Y 552.075,Z 498.011,A -85,B 0,C 180,E1 -3139.919,E2 -3139.919} C_VEL
LIN {X 0,Y 551.92,Z 505.5,A -85,B 0,C 180,E1 -3141.211,E2 -3141.211} C_VEL
LIN {X 0,Y 551.821,Z 512.504,A -85,B 0,C 180,E1 -3142.683,E2 -3142.683} C_VEL
LIN {X 0,Y 551.796,Z 518.014,A -85,B 0,C 180,E1 -3144.152,E2 -3144.152} C_VEL
LIN {X 0,Y 551.706,Z 522.179,A -85,B 0,C 180,E1 -3145.617,E2 -3145.617} C_VEL
LIN {X 0,Y 551.717,Z 525.112,A -85,B 0,C 180,E1 -3147.079,E2 -3147.079} C_VEL
LIN {X 0,Y 551.642,Z 526.878,A -85,B 0,C 180,E1 -3148.54,E2 -3148.54} C_VEL
LIN {X 0,Y 551.638,Z 527.496,A -85,B 0,C 180,E1 -3150,E2 -3150} C_VEL
LIN {X 0,Y 551.644,Z 526.939,A -85,B 0,C 180,E1 -3151.46,E2 -3151.46} C_VEL
LIN {X 0,Y 551.719,Z 525.254,A -85,B 0,C 180,E1 -3152.921,E2 -3152.921} C_VEL
LIN {X 0,Y 551.706,Z 522.401,A -85,B 0,C 180,E1 -3154.383,E2 -3154.383} C_VEL
LIN {X 0,Y 551.787,Z 518.315,A -85,B 0,C 180,E1 -3155.848,E2 -3155.848} C_VEL
LIN {X 0,Y 551.821,Z 512.898,A -85,B 0,C 180,E1 -3157.317,E2 -3157.317} C_VEL
LIN {X 0,Y 551.919,Z 505.996,A -85,B 0,C 180,E1 -3158.789,E2 -3158.789} C_VEL
LIN {X 0,Y 552.071,Z 498.571,A -85,B 0,C 180,E1 -3160.081,E2 -3160.081} C_VEL
LIN {X 0,Y 552.183,Z 490.06,A -85,B 0,C 180,E1 -3161.32,E2 -3161.32} C_VEL
LIN {X 0,Y 552.403,Z 480.533,A -85,B 0,C 180,E1 -3162.491,E2 -3162.491} C_VEL
LIN {X 0,Y 552.672,Z 469.798,A -85,B 0,C 180,E1 -3163.606,E2 -3163.606} C_VEL
LIN {X 0,Y 552.969,Z 458.085,A -85,B 0,C 180,E1 -3164.631,E2 -3164.631} C_VEL
LIN {X 0,Y 553.294,Z 445.301,A -85,B 0,C 180,E1 -3165.565,E2 -3165.565} C_VEL
LIN {X 0,Y 553.629,Z 432.971,A -85,B 0,C 180,E1 -3166.311,E2 -3166.311} C_VEL
LIN {X 0,Y 553.906,Z 418.676,A -85,B 0,C 180,E1 -3167.014,E2 -3167.014} C_VEL
LIN {X 0,Y 554.149,Z 403.818,A -85,B 0,C 180,E1 -3167.577,E2 -3167.577} C_VEL
LIN {X 0,Y 554.403,Z 388.629,A -85,B 0,C 180,E1 -3167.991,E2 -3167.991} C_VEL
LIN {X 0,Y 554.529,Z 371.968,A -85,B 0,C 180,E1 -3168.278,E2 -3168.278} C_VEL
LIN {X 0,Y 555.165,Z 227.354,A -85,B 0,C 180,E1 -3170.198,E2 -3170.198} C_VEL
LIN {X 0,Y 553.109,Z 217.125,A -85,B 0,C 180,E1 -3170.437,E2 -3170.437} C_VEL
LIN {X 0,Y 553.492,Z 200.978,A -85,B 0,C 180,E1 -3172.785,E2 -3172.785} C_VEL
LIN {X 0,Y 552.537,Z 195.242,A -85,B 0,C 180,E1 -3173.68,E2 -3173.68} C_VEL
LIN {X 0,Y 552.13,Z 193.337,A -85,B 0,C 180,E1 -3174.006,E2 -3174.006} C_VEL
LIN {X 0,Y 552.12,Z 193.334,A -85,B 0,C 180,E1 -3176.456,E2 -3176.456} C_VEL
LIN {X 0,Y 552.109,Z 193.335,A -85,B 0,C 180,E1 -3178.928,E2 -3178.928} C_VEL
LIN {X 0,Y 552.109,Z 193.341,A -85,B 0,C 180,E1 -3181.475,E2 -3181.475} C_VEL
LIN {X 0,Y 552.134,Z 193.33,A -85,B 0,C 180,E1 -3184.17,E2 -3184.17} C_VEL
LIN {X 0,Y 552.106,Z 193.334,A -85,B 0,C 180,E1 -3186.746,E2 -3186.746} C_VEL
LIN {X 0,Y 552.13,Z 193.336,A -85,B 0,C 180,E1 -3189.526,E2 -3189.526} C_VEL
LIN {X 0,Y 552.127,Z 193.33,A -85,B 0,C 180,E1 -3192.425,E2 -3192.425} C_VEL
LIN {X 0,Y 552.093,Z 193.339,A -85,B 0,C 180,E1 -3195.562,E2 -3195.562} C_VEL
LIN {X 0,Y 552.135,Z 193.329,A -85,B 0,C 180,E1 -3198.675,E2 -3198.675} C_VEL
LIN {X 0,Y 552.114,Z 193.334,A -85,B 0,C 180,E1 -3201.411,E2 -3201.411} C_VEL
LIN {X 0,Y 552.107,Z 193.331,A -85,B 0,C 180,E1 -3204.158,E2 -3204.158} C_VEL
LIN {X 0,Y 552.116,Z 193.335,A -85,B 0,C 180,E1 -3206.814,E2 -3206.814} C_VEL
LIN {X 0,Y 552.107,Z 193.335,A -85,B 0,C 180,E1 -3209.391,E2 -3209.391} C_VEL
LIN {X 0,Y 552.118,Z 193.331,A -85,B 0,C 180,E1 -3211.902,E2 -3211.902} C_VEL
LIN {X 0,Y 552.147,Z 193.33,A -85,B 0,C 180,E1 -3214.649,E2 -3214.649} C_VEL
LIN {X 0,Y 552.088,Z 193.335,A -85,B 0,C 180,E1 -3217.549,E2 -3217.549} C_VEL
LIN {X 0,Y 552.14,Z 193.33,A -85,B 0,C 180,E1 -3220.373,E2 -3220.373} C_VEL
LIN {X 0,Y 552.149,Z 193.335,A -85,B 0,C 180,E1 -3222.977,E2 -3222.977} C_VEL
LIN {X 0,Y 552.128,Z 193.327,A -85,B 0,C 180,E1 -3226.004,E2 -3226.004} C_VEL
LIN {X 0,Y 552.169,Z 193.33,A -85,B 0,C 180,E1 -3228.993,E2 -3228.993} C_VEL
LIN {X 0,Y 552.152,Z 193.326,A -85,B 0,C 180,E1 -3231.951,E2 -3231.951} C_VEL
LIN {X 0,Y 552.225,Z 193.324,A -85,B 0,C 180,E1 -3234.889,E2 -3234.889} C_VEL
LIN {X 0,Y 552.212,Z 193.319,A -85,B 0,C 180,E1 -3237.812,E2 -3237.812} C_VEL
LIN {X 0,Y 552.239,Z 193.324,A -85,B 0,C 180,E1 -3240.729,E2 -3240.729} C_VEL
LIN {X 0,Y 552.202,Z 193.324,A -85,B 0,C 180,E1 -3242.918,E2 -3242.918} C_VEL
LIN {X 0,Y 552.191,Z 193.322,A -85,B 0,C 180,E1 -3245.844,E2 -3245.844} C_VEL
LIN {X 0,Y 552.162,Z 193.33,A -85,B 0,C 180,E1 -3248.786,E2 -3248.786} C_VEL
LIN {X 0,Y 552.155,Z 193.327,A -85,B 0,C 180,E1 -3251.751,E2 -3251.751} C_VEL
LIN {X 0,Y 552.127,Z 193.335,A -85,B 0,C 180,E1 -3254.749,E2 -3254.749} C_VEL
LIN {X 0,Y 552.106,Z 193.332,A -85,B 0,C 180,E1 -3257.789,E2 -3257.789} C_VEL
LIN {X 0,Y 552.125,Z 193.336,A -85,B 0,C 180,E1 -3260.101,E2 -3260.101} C_VEL
LIN {X 0,Y 552.088,Z 193.343,A -85,B 0,C 180,E1 -3262.451,E2 -3262.451} C_VEL
LIN {X 0,Y 552.146,Z 193.326,A -85,B 0,C 180,E1 -3265.351,E2 -3265.351} C_VEL
LIN {X 0,Y 552.118,Z 193.338,A -85,B 0,C 180,E1 -3268.098,E2 -3268.098} C_VEL
LIN {X 0,Y 552.106,Z 193.336,A -85,B 0,C 180,E1 -3270.609,E2 -3270.609} C_VEL
LIN {X 0,Y 552.115,Z 193.33,A -85,B 0,C 180,E1 -3273.186,E2 -3273.186} C_VEL
LIN {X 0,Y 552.106,Z 193.337,A -85,B 0,C 180,E1 -3275.842,E2 -3275.842} C_VEL
LIN {X 0,Y 552.116,Z 193.33,A -85,B 0,C 180,E1 -3279.062,E2 -3279.062} C_VEL
LIN {X 0,Y 552.133,Z 193.327,A -85,B 0,C 180,E1 -3281.445,E2 -3281.445} C_VEL
LIN {X 0,Y 552.089,Z 193.337,A -85,B 0,C 180,E1 -3284.532,E2 -3284.532} C_VEL
LIN {X 0,Y 552.126,Z 193.333,A -85,B 0,C 180,E1 -3287.585,E2 -3287.585} C_VEL
LIN {X 0,Y 552.129,Z 193.332,A -85,B 0,C 180,E1 -3290.474,E2 -3290.474} C_VEL
LIN {X 0,Y 552.108,Z 193.333,A -85,B 0,C 180,E1 -3293.317,E2 -3293.317} C_VEL
LIN {X 0,Y 552.125,Z 193.339,A -85,B 0,C 180,E1 -3295.94,E2 -3295.94} C_VEL
LIN {X 0,Y 552.116,Z 193.332,A -85,B 0,C 180,E1 -3298.541,E2 -3298.541} C_VEL
LIN {X 0,Y 552.122,Z 193.337,A -85,B 0,C 180,E1 -3301.439,E2 -3301.439} C_VEL
LIN {X 0,Y 552.139,Z 193.505,A -85,B 0,C 180,E1 -3303,E2 -3303} C_VEL
LIN {X 0,Y 554.087,Z 202.347,A -85,B 0,C 180,E1 -3304.231,E2 -3304.231} C_VEL
LIN {X 0,Y 553.713,Z 223.006,A -85,B 0,C 180,E1 -3306.83,E2 -3306.83} C_VEL
LIN {X 0,Y 553.302,Z 245.57,A -85,B 0,C 180,E1 -3309.615,E2 -3309.615} C_VEL
LIN {X 0,Y 555.129,Z 255.497,A -85,B 0,C 180,E1 -3309.827,E2 -3309.827} C_VEL
LIN {X 0,Y 554.467,Z 412.088,A -85,B 0,C 180,E1 -3311.923,E2 -3311.923} C_VEL
LIN {X 0,Y 554.293,Z 427.686,A -85,B 0,C 180,E1 -3312.284,E2 -3312.284} C_VEL
LIN {X 0,Y 554.014,Z 443.042,A -85,B 0,C 180,E1 -3312.799,E2 -3312.799} C_VEL
LIN {X 0,Y 553.742,Z 456.79,A -85,B 0,C 180,E1 -3313.408,E2 -3313.408} C_VEL
LIN {X 0,Y 553.415,Z 470.26,A -85,B 0,C 180,E1 -3314.155,E2 -3314.155} C_VEL
LIN {X 0,Y 553.077,Z 484.151,A -85,B 0,C 180,E1 -3315.103,E2 -3315.103} C_VEL
LIN {X 0,Y 552.76,Z 496.359,A -85,B 0,C 180,E1 -3316.115,E2 -3316.115} C_VEL
LIN {X 0,Y 552.481,Z 508.511,A -85,B 0,C 180,E1 -3317.325,E2 -3317.325} C_VEL
LIN {X 0,Y 552.215,Z 518.485,A -85,B 0,C 180,E1 -3318.514,E2 -3318.514} C_VEL
LIN {X 0,Y 552.124,Z 527.087,A -85,B 0,C 180,E1 -3319.735,E2 -3319.735} C_VEL
LIN {X 0,Y 551.921,Z 534.743,A -85,B 0,C 180,E1 -3321.026,E2 -3321.026} C_VEL
LIN {X 0,Y 551.837,Z 541.09,A -85,B 0,C 180,E1 -3322.315,E2 -3322.315} C_VEL
LIN {X 0,Y 551.769,Z 546.57,A -85,B 0,C 180,E1 -3323.681,E2 -3323.681} C_VEL
LIN {X 0,Y 551.713,Z 550.387,A -85,B 0,C 180,E1 -3324.884,E2 -3324.884} C_VEL
LIN {X 0,Y 551.73,Z 553.888,A -85,B 0,C 180,E1 -3326.348,E2 -3326.348} C_VEL
LIN {X 0,Y 551.655,Z 556.19,A -85,B 0,C 180,E1 -3327.81,E2 -3327.81} C_VEL
LIN {X 0,Y 551.639,Z 557.348,A -85,B 0,C 180,E1 -3329.27,E2 -3329.27} C_VEL
LIN {X 0,Y 551.639,Z 557.347,A -85,B 0,C 180,E1 -3330.73,E2 -3330.73} C_VEL
LIN {X 0,Y 551.655,Z 556.187,A -85,B 0,C 180,E1 -3332.19,E2 -3332.19} C_VEL
LIN {X 0,Y 551.73,Z 553.884,A -85,B 0,C 180,E1 -3333.652,E2 -3333.652} C_VEL
LIN {X 0,Y 551.713,Z 550.387,A -85,B 0,C 180,E1 -3335.116,E2 -3335.116} C_VEL
LIN {X 0,Y 551.82,Z 545.61,A -85,B 0,C 180,E1 -3336.582,E2 -3336.582} C_VEL
LIN {X 0,Y 551.876,Z 539.421,A -85,B 0,C 180,E1 -3338.052,E2 -3338.052} C_VEL
LIN {X 0,Y 551.95,Z 531.645,A -85,B 0,C 180,E1 -3339.528,E2 -3339.528} C_VEL
LIN {X 0,Y 552.184,Z 523.369,A -85,B 0,C 180,E1 -3340.82,E2 -3340.82} C_VEL
LIN {X 0,Y 552.352,Z 513.393,A -85,B 0,C 180,E1 -3342.119,E2 -3342.119} C_VEL
LIN {X 0,Y 552.608,Z 503.187,A -85,B 0,C 180,E1 -3343.233,E2 -3343.233} C_VEL
LIN {X 0,Y 552.907,Z 491.022,A -85,B 0,C 180,E1 -3344.351,E2 -3344.351} C_VEL
LIN {X 0,Y 553.249,Z 478.444,A -85,B 0,C 180,E1 -3345.309,E2 -3345.309} C_VEL
LIN {X 0,Y 553.555,Z 465.51,A -85,B 0,C 180,E1 -3346.124,E2 -3346.124} C_VEL
LIN {X 0,Y 553.875,Z 450.828,A -85,B 0,C 180,E1 -3346.873,E2 -3346.873} C_VEL
LIN {X 0,Y 554.159,Z 436.616,A -85,B 0,C 180,E1 -3347.434,E2 -3347.434} C_VEL
LIN {X 0,Y 554.352,Z 421.485,A -85,B 0,C 180,E1 -3347.877,E2 -3347.877} C_VEL
LIN {X 0,Y 554.514,Z 406.098,A -85,B 0,C 180,E1 -3348.171,E2 -3348.171} C_VEL
LIN {X 0,Y 555.14,Z 255.191,A -85,B 0,C 180,E1 -3350.177,E2 -3350.177} C_VEL
LIN {X 0,Y 553.33,Z 245.56,A -85,B 0,C 180,E1 -3350.386,E2 -3350.386} C_VEL
LIN {X 0,Y 553.797,Z 219.86,A -85,B 0,C 180,E1 -3353.562,E2 -3353.562} C_VEL
LIN {X 0,Y 554.076,Z 202.375,A -85,B 0,C 180,E1 -3355.766,E2 -3355.766} C_VEL
LIN {X 0,Y 552.12,Z 193.336,A -85,B 0,C 180,E1 -3357.055,E2 -3357.055} C_VEL
LIN {X 0,Y 552.114,Z 193.338,A -85,B 0,C 180,E1 -3360.05,E2 -3360.05} C_VEL
LIN {X 0,Y 552.125,Z 193.328,A -85,B 0,C 180,E1 -3362.848,E2 -3362.848} C_VEL
LIN {X 0,Y 552.09,Z 193.334,A -85,B 0,C 180,E1 -3365.442,E2 -3365.442} C_VEL
LIN {X 0,Y 552.094,Z 193.341,A -85,B 0,C 180,E1 -3367.885,E2 -3367.885} C_VEL
LIN {X 0,Y 552.138,Z 193.332,A -85,B 0,C 180,E1 -3370.477,E2 -3370.477} C_VEL
LIN {X 0,Y 552.113,Z 193.333,A -85,B 0,C 180,E1 -3373.484,E2 -3373.484} C_VEL
LIN {X 0,Y 552.1,Z 193.334,A -85,B 0,C 180,E1 -3376.576,E2 -3376.576} C_VEL
LIN {X 0,Y 552.136,Z 193.331,A -85,B 0,C 180,E1 -3379.521,E2 -3379.521} C_VEL
LIN {X 0,Y 552.087,Z 193.337,A -85,B 0,C 180,E1 -3382.336,E2 -3382.336} C_VEL
LIN {X 0,Y 552.122,Z 193.329,A -85,B 0,C 180,E1 -3385.054,E2 -3385.054} C_VEL
LIN {X 0,Y 552.12,Z 193.336,A -85,B 0,C 180,E1 -3387.682,E2 -3387.682} C_VEL
LIN {X 0,Y 552.137,Z 193.33,A -85,B 0,C 180,E1 -3390.237,E2 -3390.237} C_VEL
LIN {X 0,Y 552.133,Z 193.329,A -85,B 0,C 180,E1 -3392.999,E2 -3392.999} C_VEL
LIN {X 0,Y 552.104,Z 193.334,A -85,B 0,C 180,E1 -3395.161,E2 -3395.161} C_VEL
LIN {X 0,Y 552.088,Z 193.34,A -85,B 0,C 180,E1 -3397.549,E2 -3397.549} C_VEL
LIN {X 0,Y 552.14,Z 193.328,A -85,B 0,C 180,E1 -3400.373,E2 -3400.373} C_VEL
LIN {X 0,Y 552.149,Z 193.328,A -85,B 0,C 180,E1 -3402.977,E2 -3402.977} C_VEL
LIN {X 0,Y 552.128,Z 193.332,A -85,B 0,C 180,E1 -3406.004,E2 -3406.004} C_VEL
LIN {X 0,Y 552.169,Z 193.326,A -85,B 0,C 180,E1 -3408.994,E2 -3408.994} C_VEL
LIN {X 0,Y 552.155,Z 193.328,A -85,B 0,C 180,E1 -3411.952,E2 -3411.952} C_VEL
LIN {X 0,Y 552.226,Z 193.319,A -85,B 0,C 180,E1 -3414.889,E2 -3414.889} C_VEL
LIN {X 0,Y 552.213,Z 193.322,A -85,B 0,C 180,E1 -3417.812,E2 -3417.812} C_VEL
LIN {X 0,Y 552.238,Z 193.315,A -85,B 0,C 180,E1 -3420.729,E2 -3420.729} C_VEL
LIN {X 0,Y 552.202,Z 193.323,A -85,B 0,C 180,E1 -3422.918,E2 -3422.918} C_VEL
LIN {X 0,Y 552.192,Z 193.323,A -85,B 0,C 180,E1 -3425.844,E2 -3425.844} C_VEL
LIN {X 0,Y 552.163,Z 193.326,A -85,B 0,C 180,E1 -3428.786,E2 -3428.786} C_VEL
LIN {X 0,Y 552.156,Z 193.327,A -85,B 0,C 180,E1 -3431.751,E2 -3431.751} C_VEL
LIN {X 0,Y 552.127,Z 193.332,A -85,B 0,C 180,E1 -3434.749,E2 -3434.749} C_VEL
LIN {X 0,Y 552.106,Z 193.333,A -85,B 0,C 180,E1 -3437.789,E2 -3437.789} C_VEL
LIN {X 0,Y 552.122,Z 193.329,A -85,B 0,C 180,E1 -3440.102,E2 -3440.102} C_VEL
LIN {X 0,Y 552.087,Z 193.336,A -85,B 0,C 180,E1 -3442.451,E2 -3442.451} C_VEL
LIN {X 0,Y 552.147,Z 193.326,A -85,B 0,C 180,E1 -3445.351,E2 -3445.351} C_VEL
LIN {X 0,Y 552.118,Z 193.33,A -85,B 0,C 180,E1 -3448.098,E2 -3448.098} C_VEL
LIN {X 0,Y 552.106,Z 193.336,A -85,B 0,C 180,E1 -3450.624,E2 -3450.624} C_VEL
LIN {X 0,Y 552.116,Z 193.335,A -85,B 0,C 180,E1 -3453.186,E2 -3453.186} C_VEL
LIN {X 0,Y 552.109,Z 193.331,A -85,B 0,C 180,E1 -3453.804,E2 -3453.804} C_VEL
LIN {X 0,Y 551.474,Z 193.413,A -85,B 0,C 180,E1 -3454.412,E2 -3454.412} C_VEL
LIN {X 0,Y 548.652,Z 193.771,A -85,B 0,C 180,E1 -3455.4,E2 -3455.4} C_VEL
LIN {X 0,Y 546.23,Z 194.076,A -85,B 0,C 180,E1 -3456.196,E2 -3456.196} C_VEL
LIN {X 0,Y 545.161,Z 194.206,A -85,B 0,C 180,E1 -3456.81,E2 -3456.81} C_VEL
LIN {X 0,Y 545.059,Z 194.216,A -85,B 0,C 180,E1 -3457.018,E2 -3457.018} C_VEL
LIN {X 0,Y 545.069,Z 194.208,A -85,B 0,C 180,E1 -3460.142,E2 -3460.142} C_VEL
LIN {X 0,Y 545.073,Z 194.212,A -85,B 0,C 180,E1 -3463.107,E2 -3463.107} C_VEL
LIN {X 0,Y 545.061,Z 194.212,A -85,B 0,C 180,E1 -3466.225,E2 -3466.225} C_VEL
LIN {X 0,Y 545.09,Z 194.214,A -85,B 0,C 180,E1 -3468.887,E2 -3468.887} C_VEL
LIN {X 0,Y 545.049,Z 194.211,A -85,B 0,C 180,E1 -3471.763,E2 -3471.763} C_VEL
LIN {X 0,Y 545.034,Z 194.22,A -85,B 0,C 180,E1 -3474.532,E2 -3474.532} C_VEL
LIN {X 0,Y 545.08,Z 194.21,A -85,B 0,C 180,E1 -3477.213,E2 -3477.213} C_VEL
LIN {X 0,Y 545.063,Z 194.212,A -85,B 0,C 180,E1 -3479.811,E2 -3479.811} C_VEL
LIN {X 0,Y 545.088,Z 194.214,A -85,B 0,C 180,E1 -3482.345,E2 -3482.345} C_VEL
LIN {X 0,Y 545.117,Z 194.211,A -85,B 0,C 180,E1 -3484.821,E2 -3484.821} C_VEL
LIN {X 0,Y 545.094,Z 194.219,A -85,B 0,C 180,E1 -3485.885,E2 -3485.885} C_VEL
LIN {X 0,Y 546.629,Z 201.884,A -85,B 0,C 180,E1 -3487.113,E2 -3487.113} C_VEL
LIN {X 0,Y 546.258,Z 217.434,A -85,B 0,C 180,E1 -3489.405,E2 -3489.405} C_VEL
LIN {X 0,Y 548.518,Z 227.991,A -85,B 0,C 180,E1 -3489.643,E2 -3489.643} C_VEL
LIN {X 0,Y 547.75,Z 382.595,A -85,B 0,C 180,E1 -3491.741,E2 -3491.741} C_VEL
LIN {X 0,Y 547.534,Z 398.137,A -85,B 0,C 180,E1 -3492.107,E2 -3492.107} C_VEL
LIN {X 0,Y 547.229,Z 413.389,A -85,B 0,C 180,E1 -3492.627,E2 -3492.627} C_VEL
LIN {X 0,Y 546.933,Z 427.984,A -85,B 0,C 180,E1 -3493.291,E2 -3493.291} C_VEL
LIN {X 0,Y 546.551,Z 441.256,A -85,B 0,C 180,E1 -3494.047,E2 -3494.047} C_VEL
LIN {X 0,Y 546.178,Z 454.417,A -85,B 0,C 180,E1 -3494.966,E2 -3494.966} C_VEL
LIN {X 0,Y 545.786,Z 466.969,A -85,B 0,C 180,E1 -3496.029,E2 -3496.029} C_VEL
LIN {X 0,Y 545.525,Z 478.104,A -85,B 0,C 180,E1 -3497.16,E2 -3497.16} C_VEL
LIN {X 0,Y 545.205,Z 488.659,A -85,B 0,C 180,E1 -3498.431,E2 -3498.431} C_VEL
LIN {X 0,Y 545.05,Z 498.014,A -85,B 0,C 180,E1 -3499.788,E2 -3499.788} C_VEL
LIN {X 0,Y 544.846,Z 505.502,A -85,B 0,C 180,E1 -3501.096,E2 -3501.096} C_VEL
LIN {X 0,Y 544.746,Z 512.506,A -85,B 0,C 180,E1 -3502.588,E2 -3502.588} C_VEL
LIN {X 0,Y 544.708,Z 518.016,A -85,B 0,C 180,E1 -3504.076,E2 -3504.076} C_VEL
LIN {X 0,Y 544.605,Z 522.18,A -85,B 0,C 180,E1 -3505.559,E2 -3505.559} C_VEL
LIN {X 0,Y 544.643,Z 525.112,A -85,B 0,C 180,E1 -3507.041,E2 -3507.041} C_VEL
LIN {X 0,Y 544.543,Z 526.878,A -85,B 0,C 180,E1 -3508.521,E2 -3508.521} C_VEL
LIN {X 0,Y 544.539,Z 527.496,A -85,B 0,C 180,E1 -3510,E2 -3510} C_VEL
LIN {X 0,Y 544.545,Z 526.938,A -85,B 0,C 180,E1 -3511.479,E2 -3511.479} C_VEL
LIN {X 0,Y 544.645,Z 525.252,A -85,B 0,C 180,E1 -3512.959,E2 -3512.959} C_VEL
LIN {X 0,Y 544.605,Z 522.399,A -85,B 0,C 180,E1 -3514.441,E2 -3514.441} C_VEL
LIN {X 0,Y 544.696,Z 518.313,A -85,B 0,C 180,E1 -3515.925,E2 -3515.925} C_VEL
LIN {X 0,Y 544.746,Z 512.895,A -85,B 0,C 180,E1 -3517.412,E2 -3517.412} C_VEL
LIN {X 0,Y 544.845,Z 505.993,A -85,B 0,C 180,E1 -3518.904,E2 -3518.904} C_VEL
LIN {X 0,Y 545.081,Z 497.38,A -85,B 0,C 180,E1 -3520.399,E2 -3520.399} C_VEL
LIN {X 0,Y 545.226,Z 488.102,A -85,B 0,C 180,E1 -3521.729,E2 -3521.729} C_VEL
LIN {X 0,Y 545.491,Z 478.9,A -85,B 0,C 180,E1 -3522.841,E2 -3522.841} C_VEL
LIN {X 0,Y 545.817,Z 466.909,A -85,B 0,C 180,E1 -3524.065,E2 -3524.065} C_VEL
LIN {X 0,Y 546.171,Z 454.963,A -85,B 0,C 180,E1 -3525.08,E2 -3525.08} C_VEL
LIN {X 0,Y 546.535,Z 441.168,A -85,B 0,C 180,E1 -3526.049,E2 -3526.049} C_VEL
LIN {X 0,Y 546.908,Z 427.881,A -85,B 0,C 180,E1 -3526.806,E2 -3526.806} C_VEL
LIN {X 0,Y 547.241,Z 413.228,A -85,B 0,C 180,E1 -3527.469,E2 -3527.469} C_VEL
LIN {X 0,Y 547.543,Z 398.523,A -85,B 0,C 180,E1 -3527.97,E2 -3527.97} C_VEL
LIN {X 0,Y 547.733,Z 383.688,A -85,B 0,C 180,E1 -3528.327,E2 -3528.327} C_VEL
LIN {X 0,Y 547.929,Z 348.664,A -85,B 0,C 180,E1 -3528.824,E2 -3528.824} C_VEL
LIN {X 0,Y 548.372,Z 227.005,A -85,B 0,C 180,E1 -3530.467,E2 -3530.467} C_VEL
LIN {X 0,Y 546.279,Z 217.312,A -85,B 0,C 180,E1 -3530.704,E2 -3530.704} C_VEL
LIN {X 0,Y 546.645,Z 202.486,A -85,B 0,C 180,E1 -3532.886,E2 -3532.886} C_VEL
LIN {X 0,Y 545.321,Z 195.266,A -85,B 0,C 180,E1 -3534.036,E2 -3534.036} C_VEL
LIN {X 0,Y 545.091,Z 194.213,A -85,B 0,C 180,E1 -3534.206,E2 -3534.206} C_VEL
LIN {X 0,Y 545.092,Z 194.214,A -85,B 0,C 180,E1 -3537.173,E2 -3537.173} C_VEL
LIN {X 0,Y 545.064,Z 194.217,A -85,B 0,C 180,E1 -3539.338,E2 -3539.338} C_VEL
LIN {X 0,Y 545.058,Z 194.215,A -85,B 0,C 180,E1 -3541.914,E2 -3541.914} C_VEL
LIN {X 0,Y 545.075,Z 194.209,A -85,B 0,C 180,E1 -3544.563,E2 -3544.563} C_VEL
LIN {X 0,Y 545.035,Z 194.22,A -85,B 0,C 180,E1 -3547.303,E2 -3547.303} C_VEL
LIN {X 0,Y 545.071,Z 194.209,A -85,B 0,C 180,E1 -3550.141,E2 -3550.141} C_VEL
LIN {X 0,Y 545.083,Z 194.213,A -85,B 0,C 180,E1 -3553.105,E2 -3553.105} C_VEL
LIN {X 0,Y 545.062,Z 194.209,A -85,B 0,C 180,E1 -3556.223,E2 -3556.223} C_VEL
LIN {X 0,Y 545.096,Z 194.208,A -85,B 0,C 180,E1 -3558.887,E2 -3558.887} C_VEL
LIN {X 0,Y 545.048,Z 194.21,A -85,B 0,C 180,E1 -3561.762,E2 -3561.762} C_VEL
LIN {X 0,Y 545.059,Z 194.21,A -85,B 0,C 180,E1 -3564.533,E2 -3564.533} C_VEL
LIN {X 0,Y 545.075,Z 194.212,A -85,B 0,C 180,E1 -3567.212,E2 -3567.212} C_VEL
LIN {X 0,Y 545.095,Z 194.204,A -85,B 0,C 180,E1 -3569.812,E2 -3569.812} C_VEL
LIN {X 0,Y 545.088,Z 194.213,A -85,B 0,C 180,E1 -3572.825,E2 -3572.825} C_VEL
LIN {X 0,Y 545.044,Z 194.213,A -85,B 0,C 180,E1 -3575.63,E2 -3575.63} C_VEL
LIN {X 0,Y 545.061,Z 194.216,A -85,B 0,C 180,E1 -3578.836,E2 -3578.836} C_VEL
LIN {X 0,Y 545.076,Z 194.212,A -85,B 0,C 180,E1 -3581.195,E2 -3581.195} C_VEL
LIN {X 0,Y 545.069,Z 194.21,A -85,B 0,C 180,E1 -3583.521,E2 -3583.521} C_VEL
LIN {X 0,Y 545.087,Z 194.204,A -85,B 0,C 180,E1 -3585.82,E2 -3585.82} C_VEL
LIN {X 0,Y 545.123,Z 194.21,A -85,B 0,C 180,E1 -3588.849,E2 -3588.849} C_VEL
LIN {X 0,Y 545.122,Z 194.202,A -85,B 0,C 180,E1 -3591.847,E2 -3591.847} C_VEL
LIN {X 0,Y 545.2,Z 194.199,A -85,B 0,C 180,E1 -3594.823,E2 -3594.823} C_VEL
LIN {X 0,Y 545.184,Z 194.194,A -85,B 0,C 180,E1 -3597.784,E2 -3597.784} C_VEL
LIN {X 0,Y 545.208,Z 194.2,A -85,B 0,C 180,E1 -3600.739,E2 -3600.739} C_VEL
LIN {X 0,Y 545.168,Z 194.199,A -85,B 0,C 180,E1 -3602.956,E2 -3602.956} C_VEL
LIN {X 0,Y 545.162,Z 194.198,A -85,B 0,C 180,E1 -3605.92,E2 -3605.92} C_VEL
LIN {X 0,Y 545.119,Z 194.206,A -85,B 0,C 180,E1 -3608.9,E2 -3608.9} C_VEL
LIN {X 0,Y 545.126,Z 194.203,A -85,B 0,C 180,E1 -3611.904,E2 -3611.904} C_VEL
LIN {X 0,Y 545.076,Z 194.211,A -85,B 0,C 180,E1 -3614.944,E2 -3614.944} C_VEL
LIN {X 0,Y 545.074,Z 194.21,A -85,B 0,C 180,E1 -3618.026,E2 -3618.026} C_VEL
LIN {X 0,Y 545.09,Z 194.215,A -85,B 0,C 180,E1 -3620.372,E2 -3620.372} C_VEL
LIN {X 0,Y 545.083,Z 194.208,A -85,B 0,C 180,E1 -3623.559,E2 -3623.559} C_VEL
LIN {X 0,Y 545.072,Z 194.212,A -85,B 0,C 180,E1 -3626.001,E2 -3626.001} C_VEL
LIN {X 0,Y 545.084,Z 194.21,A -85,B 0,C 180,E1 -3628.749,E2 -3628.749} C_VEL
LIN {X 0,Y 545.07,Z 194.211,A -85,B 0,C 180,E1 -3631.683,E2 -3631.683} C_VEL
LIN {X 0,Y 545.074,Z 194.212,A -85,B 0,C 180,E1 -3634.564,E2 -3634.564} C_VEL
LIN {X 0,Y 545.032,Z 194.213,A -85,B 0,C 180,E1 -3637.304,E2 -3637.304} C_VEL
LIN {X 0,Y 545.066,Z 194.212,A -85,B 0,C 180,E1 -3640.142,E2 -3640.142} C_VEL
LIN {X 0,Y 545.056,Z 194.212,A -85,B 0,C 180,E1 -3642.697,E2 -3642.697} C_VEL
LIN {X 0,Y 545.057,Z 194.211,A -85,B 0,C 180,E1 -3645.168,E2 -3645.168} C_VEL
LIN {X 0,Y 545.078,Z 194.216,A -85,B 0,C 180,E1 -3647.898,E2 -3647.898} C_VEL
LIN {X 0,Y 545.101,Z 194.206,A -85,B 0,C 180,E1 -3650.677,E2 -3650.677} C_VEL
LIN {X 0,Y 545.046,Z 194.216,A -85,B 0,C 180,E1 -3653.621,E2 -3653.621} C_VEL
LIN {X 0,Y 545.066,Z 194.214,A -85,B 0,C 180,E1 -3656.329,E2 -3656.329} C_VEL
LIN {X 0,Y 545.063,Z 194.21,A -85,B 0,C 180,E1 -3658.953,E2 -3658.953} C_VEL
LIN {X 0,Y 545.098,Z 194.213,A -85,B 0,C 180,E1 -3661.508,E2 -3661.508} C_VEL
LIN {X 0,Y 545.117,Z 194.391,A -85,B 0,C 180,E1 -3662.765,E2 -3662.765} C_VEL
LIN {X 0,Y 547.231,Z 203.899,A -85,B 0,C 180,E1 -3664.11,E2 -3664.11} C_VEL
LIN {X 0,Y 546.875,Z 222.823,A -85,B 0,C 180,E1 -3666.523,E2 -3666.523} C_VEL
LIN {X 0,Y 546.407,Z 245.446,A -85,B 0,C 180,E1 -3669.355,E2 -3669.355} C_VEL
LIN {X 0,Y 548.476,Z 257.219,A -85,B 0,C 180,E1 -3669.598,E2 -3669.598} C_VEL
LIN {X 0,Y 547.711,Z 412.335,A -85,B 0,C 180,E1 -3671.701,E2 -3671.701} C_VEL
LIN {X 0,Y 547.524,Z 427.485,A -85,B 0,C 180,E1 -3672.058,E2 -3672.058} C_VEL
LIN {X 0,Y 547.22,Z 442.848,A -85,B 0,C 180,E1 -3672.579,E2 -3672.579} C_VEL
LIN {X 0,Y 546.898,Z 456.638,A -85,B 0,C 180,E1 -3673.194,E2 -3673.194} C_VEL
LIN {X 0,Y 546.567,Z 470.155,A -85,B 0,C 180,E1 -3673.952,E2 -3673.952} C_VEL
LIN {X 0,Y 546.143,Z 484.107,A -85,B 0,C 180,E1 -3674.91,E2 -3674.91} C_VEL
LIN {X 0,Y 545.817,Z 496.36,A -85,B 0,C 180,E1 -3675.935,E2 -3675.935} C_VEL
LIN {X 0,Y 545.511,Z 508.511,A -85,B 0,C 180,E1 -3677.16,E2 -3677.16} C_VEL
LIN {X 0,Y 545.174,Z 519.107,A -85,B 0,C 180,E1 -3678.446,E2 -3678.446} C_VEL
LIN {X 0,Y 545.05,Z 528.298,A -85,B 0,C 180,E1 -3679.788,E2 -3679.788} C_VEL
LIN {X 0,Y 544.845,Z 535.75,A -85,B 0,C 180,E1 -3681.096,E2 -3681.096} C_VEL
LIN {X 0,Y 544.744,Z 542.701,A -85,B 0,C 180,E1 -3682.588,E2 -3682.588} C_VEL
LIN {X 0,Y 544.709,Z 548.163,A -85,B 0,C 180,E1 -3684.076,E2 -3684.076} C_VEL
LIN {X 0,Y 544.605,Z 552.291,A -85,B 0,C 180,E1 -3685.559,E2 -3685.559} C_VEL
LIN {X 0,Y 544.644,Z 555.184,A -85,B 0,C 180,E1 -3687.041,E2 -3687.041} C_VEL
LIN {X 0,Y 544.544,Z 556.909,A -85,B 0,C 180,E1 -3688.521,E2 -3688.521} C_VEL
LIN {X 0,Y 544.538,Z 557.5,A -85,B 0,C 180,E1 -3690,E2 -3690} C_VEL
LIN {X 0,Y 544.544,Z 556.907,A -85,B 0,C 180,E1 -3691.479,E2 -3691.479} C_VEL
LIN {X 0,Y 544.644,Z 555.18,A -85,B 0,C 180,E1 -3692.959,E2 -3692.959} C_VEL
LIN {X 0,Y 544.605,Z 552.289,A -85,B 0,C 180,E1 -3694.441,E2 -3694.441} C_VEL
LIN {X 0,Y 544.709,Z 548.166,A -85,B 0,C 180,E1 -3695.924,E2 -3695.924} C_VEL
LIN {X 0,Y 544.745,Z 542.701,A -85,B 0,C 180,E1 -3697.412,E2 -3697.412} C_VEL
LIN {X 0,Y 544.845,Z 535.745,A -85,B 0,C 180,E1 -3698.904,E2 -3698.904} C_VEL
LIN {X 0,Y 545.074,Z 527.082,A -85,B 0,C 180,E1 -3700.399,E2 -3700.399} C_VEL
LIN {X 0,Y 545.236,Z 517.707,A -85,B 0,C 180,E1 -3701.734,E2 -3701.734} C_VEL
LIN {X 0,Y 545.511,Z 508.51,A -85,B 0,C 180,E1 -3702.84,E2 -3702.84} C_VEL
LIN {X 0,Y 545.827,Z 496.365,A -85,B 0,C 180,E1 -3704.065,E2 -3704.065} C_VEL
LIN {X 0,Y 546.17,Z 483.766,A -85,B 0,C 180,E1 -3705.115,E2 -3705.115} C_VEL
LIN {X 0,Y 546.562,Z 470.152,A -85,B 0,C 180,E1 -3706.049,E2 -3706.049} C_VEL
LIN {X 0,Y 546.924,Z 456.63,A -85,B 0,C 180,E1 -3706.805,E2 -3706.805} C_VEL
LIN {X 0,Y 547.209,Z 442.857,A -85,B 0,C 180,E1 -3707.422,E2 -3707.422} C_VEL
LIN {X 0,Y 547.513,Z 427.502,A -85,B 0,C 180,E1 -3707.942,E2 -3707.942} C_VEL
LIN {X 0,Y 547.72,Z 411.847,A -85,B 0,C 180,E1 -3708.308,E2 -3708.308} C_VEL
LIN {X 0,Y 548.489,Z 256.388,A -85,B 0,C 180,E1 -3710.413,E2 -3710.413} C_VEL
LIN {X 0,Y 546.408,Z 245.367,A -85,B 0,C 180,E1 -3710.656,E2 -3710.656} C_VEL
LIN {X 0,Y 546.924,Z 221.431,A -85,B 0,C 180,E1 -3713.652,E2 -3713.652} C_VEL
LIN {X 0,Y 547.229,Z 203.902,A -85,B 0,C 180,E1 -3715.89,E2 -3715.89} C_VEL
LIN {X 0,Y 545.092,Z 194.212,A -85,B 0,C 180,E1 -3717.271,E2 -3717.271} C_VEL
LIN {X 0,Y 545.075,Z 194.215,A -85,B 0,C 180,E1 -3720.246,E2 -3720.246} C_VEL
LIN {X 0,Y 545.085,Z 194.204,A -85,B 0,C 180,E1 -3723.063,E2 -3723.063} C_VEL
LIN {X 0,Y 545.047,Z 194.214,A -85,B 0,C 180,E1 -3725.675,E2 -3725.675} C_VEL
LIN {X 0,Y 545.05,Z 194.219,A -85,B 0,C 180,E1 -3728.236,E2 -3728.236} C_VEL
LIN {X 0,Y 545.097,Z 194.206,A -85,B 0,C 180,E1 -3731.112,E2 -3731.112} C_VEL
LIN {X 0,Y 545.054,Z 194.217,A -85,B 0,C 180,E1 -3734.128,E2 -3734.128} C_VEL
LIN {X 0,Y 545.072,Z 194.208,A -85,B 0,C 180,E1 -3736.893,E2 -3736.893} C_VEL
LIN {X 0,Y 545.087,Z 194.213,A -85,B 0,C 180,E1 -3739.859,E2 -3739.859} C_VEL
LIN {X 0,Y 545.068,Z 194.208,A -85,B 0,C 180,E1 -3743.073,E2 -3743.073} C_VEL
LIN {X 0,Y 545.078,Z 194.212,A -85,B 0,C 180,E1 -3745.606,E2 -3745.606} C_VEL
LIN {X 0,Y 545.07,Z 194.21,A -85,B 0,C 180,E1 -3748.317,E2 -3748.317} C_VEL
LIN {X 0,Y 545.084,Z 194.208,A -85,B 0,C 180,E1 -3751.251,E2 -3751.251} C_VEL
LIN {X 0,Y 545.071,Z 194.214,A -85,B 0,C 180,E1 -3753.999,E2 -3753.999} C_VEL
LIN {X 0,Y 545.083,Z 194.206,A -85,B 0,C 180,E1 -3756.441,E2 -3756.441} C_VEL
LIN {X 0,Y 545.09,Z 194.21,A -85,B 0,C 180,E1 -3759.628,E2 -3759.628} C_VEL
LIN {X 0,Y 545.087,Z 194.206,A -85,B 0,C 180,E1 -3762.75,E2 -3762.75} C_VEL
LIN {X 0,Y 545.087,Z 194.212,A -85,B 0,C 180,E1 -3765.82,E2 -3765.82} C_VEL
LIN {X 0,Y 545.123,Z 194.203,A -85,B 0,C 180,E1 -3768.85,E2 -3768.85} C_VEL
LIN {X 0,Y 545.125,Z 194.205,A -85,B 0,C 180,E1 -3771.847,E2 -3771.847} C_VEL
LIN {X 0,Y 545.201,Z 194.193,A -85,B 0,C 180,E1 -3774.823,E2 -3774.823} C_VEL
LIN {X 0,Y 545.185,Z 194.198,A -85,B 0,C 180,E1 -3777.784,E2 -3777.784} C_VEL
LIN {X 0,Y 545.208,Z 194.191,A -85,B 0,C 180,E1 -3780.739,E2 -3780.739} C_VEL
LIN {X 0,Y 545.168,Z 194.2,A -85,B 0,C 180,E1 -3782.956,E2 -3782.956} C_VEL
LIN {X 0,Y 545.163,Z 194.198,A -85,B 0,C 180,E1 -3785.92,E2 -3785.92} C_VEL
LIN {X 0,Y 545.12,Z 194.205,A -85,B 0,C 180,E1 -3788.9,E2 -3788.9} C_VEL
LIN {X 0,Y 545.127,Z 194.201,A -85,B 0,C 180,E1 -3791.904,E2 -3791.904} C_VEL
LIN {X 0,Y 545.077,Z 194.213,A -85,B 0,C 180,E1 -3794.944,E2 -3794.944} C_VEL
LIN {X 0,Y 545.074,Z 194.208,A -85,B 0,C 180,E1 -3798.026,E2 -3798.026} C_VEL
LIN {X 0,Y 545.087,Z 194.206,A -85,B 0,C 180,E1 -3800.373,E2 -3800.373} C_VEL
LIN {X 0,Y 545.083,Z 194.208,A -85,B 0,C 180,E1 -3803.559,E2 -3803.559} C_VEL
LIN {X 0,Y 545.072,Z 194.201,A -85,B 0,C 180,E1 -3806.001,E2 -3806.001} C_VEL
LIN {X 0,Y 545.085,Z 194.211,A -85,B 0,C 180,E1 -3808.75,E2 -3808.75} C_VEL
LIN {X 0,Y 545.071,Z 194.209,A -85,B 0,C 180,E1 -3811.683,E2 -3811.683} C_VEL
LIN {X 0,Y 545.075,Z 194.211,A -85,B 0,C 180,E1 -3814.564,E2 -3814.564} C_VEL
LIN {X 0,Y 545.059,Z 194.216,A -85,B 0,C 180,E1 -3817.018,E2 -3817.018} C_VEL
LIN {X 0,Y 544.351,Z 194.301,A -85,B 0,C 180,E1 -3817.634,E2 -3817.634} C_VEL
LIN {X 0,Y 541.488,Z 194.66,A -85,B 0,C 180,E1 -3818.635,E2 -3818.635} C_VEL
LIN {X 0,Y 539.102,Z 194.953,A -85,B 0,C 180,E1 -3819.441,E2 -3819.441} C_VEL
LIN {X 0,Y 538.093,Z 195.077,A -85,B 0,C 180,E1 -3820.063,E2 -3820.063} C_VEL
LIN {X 0,Y 538.017,Z 195.088,A -85,B 0,C 180,E1 -3820.274,E2 -3820.274} C_VEL
LIN {X 0,Y 538.021,Z 195.093,A -85,B 0,C 180,E1 -3822.988,E2 -3822.988} C_VEL
LIN {X 0,Y 538.025,Z 195.087,A -85,B 0,C 180,E1 -3825.926,E2 -3825.926} C_VEL
LIN {X 0,Y 538.046,Z 195.087,A -85,B 0,C 180,E1 -3829.225,E2 -3829.225} C_VEL
LIN {X 0,Y 537.989,Z 195.093,A -85,B 0,C 180,E1 -3832.123,E2 -3832.123} C_VEL
LIN {X 0,Y 537.996,Z 195.096,A -85,B 0,C 180,E1 -3834.916,E2 -3834.916} C_VEL
LIN {X 0,Y 538.025,Z 195.088,A -85,B 0,C 180,E1 -3837.619,E2 -3837.619} C_VEL
LIN {X 0,Y 538.016,Z 195.094,A -85,B 0,C 180,E1 -3840.24,E2 -3840.24} C_VEL
LIN {X 0,Y 538.063,Z 195.09,A -85,B 0,C 180,E1 -3842.797,E2 -3842.797} C_VEL
LIN {X 0,Y 538.027,Z 195.171,A -85,B 0,C 180,E1 -3845.665,E2 -3845.665} C_VEL
LIN {X 0,Y 539.742,Z 203.397,A -85,B 0,C 180,E1 -3847.007,E2 -3847.007} C_VEL
LIN {X 0,Y 539.437,Z 217.72,A -85,B 0,C 180,E1 -3849.136,E2 -3849.136} C_VEL
LIN {X 0,Y 541.867,Z 229.418,A -85,B 0,C 180,E1 -3849.398,E2 -3849.398} C_VEL
LIN {X 0,Y 541.029,Z 382.827,A -85,B 0,C 180,E1 -3851.506,E2 -3851.506} C_VEL
LIN {X 0,Y 540.809,Z 398.357,A -85,B 0,C 180,E1 -3851.876,E2 -3851.876} C_VEL
LIN {X 0,Y 540.471,Z 413.604,A -85,B 0,C 180,E1 -3852.403,E2 -3852.403} C_VEL
LIN {X 0,Y 540.166,Z 426.292,A -85,B 0,C 180,E1 -3852.978,E2 -3852.978} C_VEL
LIN {X 0,Y 539.777,Z 439.901,A -85,B 0,C 180,E1 -3853.744,E2 -3853.744} C_VEL
LIN {X 0,Y 539.345,Z 452.854,A -85,B 0,C 180,E1 -3854.637,E2 -3854.637} C_VEL
LIN {X 0,Y 538.973,Z 465.065,A -85,B 0,C 180,E1 -3855.656,E2 -3855.656} C_VEL
LIN {X 0,Y 538.616,Z 476.536,A -85,B 0,C 180,E1 -3856.801,E2 -3856.801} C_VEL
LIN {X 0,Y 538.253,Z 487.325,A -85,B 0,C 180,E1 -3858.089,E2 -3858.089} C_VEL
LIN {X 0,Y 538.043,Z 496.866,A -85,B 0,C 180,E1 -3859.463,E2 -3859.463} C_VEL
LIN {X 0,Y 537.837,Z 504.518,A -85,B 0,C 180,E1 -3860.789,E2 -3860.789} C_VEL
LIN {X 0,Y 537.701,Z 510.896,A -85,B 0,C 180,E1 -3862.112,E2 -3862.112} C_VEL
LIN {X 0,Y 537.624,Z 516.256,A -85,B 0,C 180,E1 -3863.463,E2 -3863.463} C_VEL
LIN {X 0,Y 537.574,Z 520.259,A -85,B 0,C 180,E1 -3864.749,E2 -3864.749} C_VEL
LIN {X 0,Y 537.562,Z 523.795,A -85,B 0,C 180,E1 -3866.252,E2 -3866.252} C_VEL
LIN {X 0,Y 537.488,Z 526.137,A -85,B 0,C 180,E1 -3867.752,E2 -3867.752} C_VEL
LIN {X 0,Y 537.437,Z 527.337,A -85,B 0,C 180,E1 -3869.251,E2 -3869.251} C_VEL
LIN {X 0,Y 537.439,Z 527.357,A -85,B 0,C 180,E1 -3870.749,E2 -3870.749} C_VEL
LIN {X 0,Y 537.488,Z 526.237,A -85,B 0,C 180,E1 -3872.248,E2 -3872.248} C_VEL
LIN {X 0,Y 537.562,Z 523.974,A -85,B 0,C 180,E1 -3873.748,E2 -3873.748} C_VEL
LIN {X 0,Y 537.572,Z 520.513,A -85,B 0,C 180,E1 -3875.251,E2 -3875.251} C_VEL
LIN {X 0,Y 537.619,Z 515.776,A -85,B 0,C 180,E1 -3876.756,E2 -3876.756} C_VEL
LIN {X 0,Y 537.735,Z 509.639,A -85,B 0,C 180,E1 -3878.266,E2 -3878.266} C_VEL
LIN {X 0,Y 537.861,Z 501.955,A -85,B 0,C 180,E1 -3879.78,E2 -3879.78} C_VEL
LIN {X 0,Y 538.08,Z 493.776,A -85,B 0,C 180,E1 -3881.107,E2 -3881.107} C_VEL
LIN {X 0,Y 538.347,Z 483.926,A -85,B 0,C 180,E1 -3882.439,E2 -3882.439} C_VEL
LIN {X 0,Y 538.68,Z 473.823,A -85,B 0,C 180,E1 -3883.582,E2 -3883.582} C_VEL
LIN {X 0,Y 539.034,Z 461.797,A -85,B 0,C 180,E1 -3884.728,E2 -3884.728} C_VEL
LIN {X 0,Y 539.503,Z 448.469,A -85,B 0,C 180,E1 -3885.778,E2 -3885.778} C_VEL
LIN {X 0,Y 539.948,Z 435.062,A -85,B 0,C 180,E1 -3886.639,E2 -3886.639} C_VEL
LIN {X 0,Y 540.263,Z 421.194,A -85,B 0,C 180,E1 -3887.36,E2 -3887.36} C_VEL
LIN {X 0,Y 540.621,Z 405.672,A -85,B 0,C 180,E1 -3887.983,E2 -3887.983} C_VEL
LIN {X 0,Y 540.933,Z 390.113,A -85,B 0,C 180,E1 -3888.43,E2 -3888.43} C_VEL
LIN {X 0,Y 541.095,Z 373.637,A -85,B 0,C 180,E1 -3888.729,E2 -3888.729} C_VEL
LIN {X 0,Y 541.854,Z 228.741,A -85,B 0,C 180,E1 -3890.702,E2 -3890.702} C_VEL
LIN {X 0,Y 539.462,Z 217.495,A -85,B 0,C 180,E1 -3890.978,E2 -3890.978} C_VEL
LIN {X 0,Y 539.796,Z 203.993,A -85,B 0,C 180,E1 -3892.991,E2 -3892.991} C_VEL
LIN {X 0,Y 538.026,Z 195.092,A -85,B 0,C 180,E1 -3894.456,E2 -3894.456} C_VEL
LIN {X 0,Y 538.057,Z 195.091,A -85,B 0,C 180,E1 -3897.351,E2 -3897.351} C_VEL
LIN {X 0,Y 538.016,Z 195.095,A -85,B 0,C 180,E1 -3899.76,E2 -3899.76} C_VEL
LIN {X 0,Y 538.025,Z 195.088,A -85,B 0,C 180,E1 -3902.381,E2 -3902.381} C_VEL
LIN {X 0,Y 538.01,Z 195.094,A -85,B 0,C 180,E1 -3905.083,E2 -3905.083} C_VEL
LIN {X 0,Y 537.99,Z 195.095,A -85,B 0,C 180,E1 -3907.877,E2 -3907.877} C_VEL
LIN {X 0,Y 538.048,Z 195.085,A -85,B 0,C 180,E1 -3910.775,E2 -3910.775} C_VEL
LIN {X 0,Y 538.025,Z 195.087,A -85,B 0,C 180,E1 -3914.074,E2 -3914.074} C_VEL
LIN {X 0,Y 538.021,Z 195.092,A -85,B 0,C 180,E1 -3917.012,E2 -3917.012} C_VEL
LIN {X 0,Y 538.073,Z 195.088,A -85,B 0,C 180,E1 -3919.248,E2 -3919.248} C_VEL
LIN {X 0,Y 537.988,Z 195.087,A -85,B 0,C 180,E1 -3922.122,E2 -3922.122} C_VEL
LIN {X 0,Y 538.014,Z 195.092,A -85,B 0,C 180,E1 -3924.917,E2 -3924.917} C_VEL
LIN {X 0,Y 538.024,Z 195.084,A -85,B 0,C 180,E1 -3927.618,E2 -3927.618} C_VEL
LIN {X 0,Y 538.036,Z 195.083,A -85,B 0,C 180,E1 -3930.24,E2 -3930.24} C_VEL
LIN {X 0,Y 538.058,Z 195.088,A -85,B 0,C 180,E1 -3932.796,E2 -3932.796} C_VEL
LIN {X 0,Y 538.041,Z 195.089,A -85,B 0,C 180,E1 -3935.292,E2 -3935.292} C_VEL
LIN {X 0,Y 538.006,Z 195.087,A -85,B 0,C 180,E1 -3938.041,E2 -3938.041} C_VEL
LIN {X 0,Y 538.032,Z 195.092,A -85,B 0,C 180,E1 -3940.94,E2 -3940.94} C_VEL
LIN {X 0,Y 538.019,Z 195.091,A -85,B 0,C 180,E1 -3943.299,E2 -3943.299} C_VEL
LIN {X 0,Y 538.055,Z 195.081,A -85,B 0,C 180,E1 -3945.63,E2 -3945.63} C_VEL
LIN {X 0,Y 538.08,Z 195.087,A -85,B 0,C 180,E1 -3948.702,E2 -3948.702} C_VEL
LIN {X 0,Y 538.079,Z 195.079,A -85,B 0,C 180,E1 -3951.739,E2 -3951.739} C_VEL
LIN {X 0,Y 538.157,Z 195.076,A -85,B 0,C 180,E1 -3954.755,E2 -3954.755} C_VEL
LIN {X 0,Y 538.157,Z 195.07,A -85,B 0,C 180,E1 -3957.755,E2 -3957.755} C_VEL
LIN {X 0,Y 538.178,Z 195.075,A -85,B 0,C 180,E1 -3960.748,E2 -3960.748} C_VEL
LIN {X 0,Y 538.134,Z 195.075,A -85,B 0,C 180,E1 -3962.994,E2 -3962.994} C_VEL
LIN {X 0,Y 538.115,Z 195.077,A -85,B 0,C 180,E1 -3965.997,E2 -3965.997} C_VEL
LIN {X 0,Y 538.068,Z 195.083,A -85,B 0,C 180,E1 -3969.018,E2 -3969.018} C_VEL
LIN {X 0,Y 538.074,Z 195.084,A -85,B 0,C 180,E1 -3972.063,E2 -3972.063} C_VEL
LIN {X 0,Y 538.036,Z 195.087,A -85,B 0,C 180,E1 -3975.144,E2 -3975.144} C_VEL
LIN {X 0,Y 538.026,Z 195.092,A -85,B 0,C 180,E1 -3978.27,E2 -3978.27} C_VEL
LIN {X 0,Y 538.033,Z 195.089,A -85,B 0,C 180,E1 -3980.652,E2 -3980.652} C_VEL
LIN {X 0,Y 538.015,Z 195.091,A -85,B 0,C 180,E1 -3983.888,E2 -3983.888} C_VEL
LIN {X 0,Y 538.034,Z 195.094,A -85,B 0,C 180,E1 -3986.367,E2 -3986.367} C_VEL
LIN {X 0,Y 538.048,Z 195.085,A -85,B 0,C 180,E1 -3988.939,E2 -3988.939} C_VEL
LIN {X 0,Y 538.02,Z 195.092,A -85,B 0,C 180,E1 -3991.891,E2 -3991.891} C_VEL
LIN {X 0,Y 538.024,Z 195.089,A -85,B 0,C 180,E1 -3994.621,E2 -3994.621} C_VEL
LIN {X 0,Y 538.001,Z 195.089,A -85,B 0,C 180,E1 -3997.171,E2 -3997.171} C_VEL
LIN {X 0,Y 538.021,Z 195.09,A -85,B 0,C 180,E1 -3999.797,E2 -3999.797} C_VEL
LIN {X 0,Y 538.013,Z 195.089,A -85,B 0,C 180,E1 -4002.787,E2 -4002.787} C_VEL
LIN {X 0,Y 538.026,Z 195.087,A -85,B 0,C 180,E1 -4005.141,E2 -4005.141} C_VEL
LIN {X 0,Y 538.036,Z 195.091,A -85,B 0,C 180,E1 -4008.228,E2 -4008.228} C_VEL
LIN {X 0,Y 538.054,Z 195.086,A -85,B 0,C 180,E1 -4010.412,E2 -4010.412} C_VEL
LIN {X 0,Y 538.023,Z 195.086,A -85,B 0,C 180,E1 -4013.068,E2 -4013.068} C_VEL
LIN {X 0,Y 538.021,Z 195.095,A -85,B 0,C 180,E1 -4015.828,E2 -4015.828} C_VEL
LIN {X 0,Y 538.006,Z 195.091,A -85,B 0,C 180,E1 -4018.499,E2 -4018.499} C_VEL
LIN {X 0,Y 538.058,Z 195.087,A -85,B 0,C 180,E1 -4021.1,E2 -4021.1} C_VEL
LIN {X 0,Y 538.071,Z 195.174,A -85,B 0,C 180,E1 -4022.508,E2 -4022.508} C_VEL
LIN {X 0,Y 540.408,Z 205.633,A -85,B 0,C 180,E1 -4024.011,E2 -4024.011} C_VEL
LIN {X 0,Y 539.975,Z 225.785,A -85,B 0,C 180,E1 -4026.612,E2 -4026.612} C_VEL
LIN {X 0,Y 539.515,Z 245.251,A -85,B 0,C 180,E1 -4029.079,E2 -4029.079} C_VEL
LIN {X 0,Y 541.765,Z 257.026,A -85,B 0,C 180,E1 -4029.334,E2 -4029.334} C_VEL
LIN {X 0,Y 541.001,Z 411.662,A -85,B 0,C 180,E1 -4031.456,E2 -4031.456} C_VEL
LIN {X 0,Y 540.752,Z 427.284,A -85,B 0,C 180,E1 -4031.825,E2 -4031.825} C_VEL
LIN {X 0,Y 540.418,Z 442.646,A -85,B 0,C 180,E1 -4032.352,E2 -4032.352} C_VEL
LIN {X 0,Y 540.047,Z 456.435,A -85,B 0,C 180,E1 -4032.974,E2 -4032.974} C_VEL
LIN {X 0,Y 539.677,Z 469.952,A -85,B 0,C 180,E1 -4033.741,E2 -4033.741} C_VEL
LIN {X 0,Y 539.298,Z 483.119,A -85,B 0,C 180,E1 -4034.655,E2 -4034.655} C_VEL
LIN {X 0,Y 538.852,Z 496.173,A -85,B 0,C 180,E1 -4035.749,E2 -4035.749} C_VEL
LIN {X 0,Y 538.525,Z 508.394,A -85,B 0,C 180,E1 -4036.99,E2 -4036.99} C_VEL
LIN {X 0,Y 538.178,Z 518.677,A -85,B 0,C 180,E1 -4038.242,E2 -4038.242} C_VEL
LIN {X 0,Y 538.017,Z 528.298,A -85,B 0,C 180,E1 -4039.653,E2 -4039.653} C_VEL
LIN {X 0,Y 537.797,Z 535.75,A -85,B 0,C 180,E1 -4040.978,E2 -4040.978} C_VEL
LIN {X 0,Y 537.661,Z 542.7,A -85,B 0,C 180,E1 -4042.489,E2 -4042.489} C_VEL
LIN {X 0,Y 537.623,Z 548.162,A -85,B 0,C 180,E1 -4043.997,E2 -4043.997} C_VEL
LIN {X 0,Y 537.507,Z 552.29,A -85,B 0,C 180,E1 -4045.501,E2 -4045.501} C_VEL
LIN {X 0,Y 537.544,Z 555.184,A -85,B 0,C 180,E1 -4047.002,E2 -4047.002} C_VEL
LIN {X 0,Y 537.449,Z 556.909,A -85,B 0,C 180,E1 -4048.501,E2 -4048.501} C_VEL
LIN {X 0,Y 537.439,Z 557.5,A -85,B 0,C 180,E1 -4050,E2 -4050} C_VEL
LIN {X 0,Y 537.449,Z 556.907,A -85,B 0,C 180,E1 -4051.499,E2 -4051.499} C_VEL
LIN {X 0,Y 537.544,Z 555.179,A -85,B 0,C 180,E1 -4052.998,E2 -4052.998} C_VEL
LIN {X 0,Y 537.507,Z 552.288,A -85,B 0,C 180,E1 -4054.499,E2 -4054.499} C_VEL
LIN {X 0,Y 537.623,Z 548.166,A -85,B 0,C 180,E1 -4056.003,E2 -4056.003} C_VEL
LIN {X 0,Y 537.661,Z 542.701,A -85,B 0,C 180,E1 -4057.511,E2 -4057.511} C_VEL
LIN {X 0,Y 537.797,Z 535.744,A -85,B 0,C 180,E1 -4059.022,E2 -4059.022} C_VEL
LIN {X 0,Y 538.024,Z 527.081,A -85,B 0,C 180,E1 -4060.537,E2 -4060.537} C_VEL
LIN {X 0,Y 538.19,Z 518.619,A -85,B 0,C 180,E1 -4061.765,E2 -4061.765} C_VEL
LIN {X 0,Y 538.525,Z 508.393,A -85,B 0,C 180,E1 -4063.01,E2 -4063.01} C_VEL
LIN {X 0,Y 538.872,Z 496.178,A -85,B 0,C 180,E1 -4064.251,E2 -4064.251} C_VEL
LIN {X 0,Y 539.291,Z 483.168,A -85,B 0,C 180,E1 -4065.343,E2 -4065.343} C_VEL
LIN {X 0,Y 539.672,Z 469.949,A -85,B 0,C 180,E1 -4066.259,E2 -4066.259} C_VEL
LIN {X 0,Y 540.07,Z 456.427,A -85,B 0,C 180,E1 -4067.025,E2 -4067.025} C_VEL
LIN {X 0,Y 540.424,Z 442.656,A -85,B 0,C 180,E1 -4067.648,E2 -4067.648} C_VEL
LIN {X 0,Y 540.74,Z 427.301,A -85,B 0,C 180,E1 -4068.175,E2 -4068.175} C_VEL
LIN {X 0,Y 540.97,Z 411.92,A -85,B 0,C 180,E1 -4068.54,E2 -4068.54} C_VEL
LIN {X 0,Y 541.825,Z 257.878,A -85,B 0,C 180,E1 -4070.652,E2 -4070.652} C_VEL
LIN {X 0,Y 539.506,Z 245.167,A -85,B 0,C 180,E1 -4070.932,E2 -4070.932} C_VEL
LIN {X 0,Y 540.052,Z 222.636,A -85,B 0,C 180,E1 -4073.792,E2 -4073.792} C_VEL
LIN {X 0,Y 540.405,Z 205.637,A -85,B 0,C 180,E1 -4075.989,E2 -4075.989} C_VEL
LIN {X 0,Y 538.047,Z 195.091,A -85,B 0,C 180,E1 -4077.517,E2 -4077.517} C_VEL
LIN {X 0,Y 538.023,Z 195.091,A -85,B 0,C 180,E1 -4080.443,E2 -4080.443} C_VEL
LIN {X 0,Y 538.042,Z 195.081,A -85,B 0,C 180,E1 -4083.282,E2 -4083.282} C_VEL
LIN {X 0,Y 538.019,Z 195.094,A -85,B 0,C 180,E1 -4086.002,E2 -4086.002} C_VEL
LIN {X 0,Y 538.011,Z 195.09,A -85,B 0,C 180,E1 -4088.83,E2 -4088.83} C_VEL
LIN {X 0,Y 538.074,Z 195.081,A -85,B 0,C 180,E1 -4090.772,E2 -4090.772} C_VEL
LIN {X 0,Y 538.025,Z 195.094,A -85,B 0,C 180,E1 -4094.074,E2 -4094.074} C_VEL
LIN {X 0,Y 538.02,Z 195.086,A -85,B 0,C 180,E1 -4097.012,E2 -4097.012} C_VEL
LIN {X 0,Y 538.072,Z 195.08,A -85,B 0,C 180,E1 -4099.248,E2 -4099.248} C_VEL
LIN {X 0,Y 537.988,Z 195.096,A -85,B 0,C 180,E1 -4102.122,E2 -4102.122} C_VEL
LIN {X 0,Y 538.013,Z 195.086,A -85,B 0,C 180,E1 -4104.917,E2 -4104.917} C_VEL
LIN {X 0,Y 538.024,Z 195.091,A -85,B 0,C 180,E1 -4107.618,E2 -4107.618} C_VEL
LIN {X 0,Y 538.035,Z 195.087,A -85,B 0,C 180,E1 -4110.24,E2 -4110.24} C_VEL
LIN {X 0,Y 538.059,Z 195.081,A -85,B 0,C 180,E1 -4112.796,E2 -4112.796} C_VEL
LIN {X 0,Y 538.04,Z 195.088,A -85,B 0,C 180,E1 -4115.292,E2 -4115.292} C_VEL
LIN {X 0,Y 538.006,Z 195.086,A -85,B 0,C 180,E1 -4118.041,E2 -4118.041} C_VEL
LIN {X 0,Y 538.032,Z 195.086,A -85,B 0,C 180,E1 -4120.94,E2 -4120.94} C_VEL
LIN {X 0,Y 538.019,Z 195.091,A -85,B 0,C 180,E1 -4123.299,E2 -4123.299} C_VEL
LIN {X 0,Y 538.055,Z 195.091,A -85,B 0,C 180,E1 -4125.631,E2 -4125.631} C_VEL
LIN {X 0,Y 538.08,Z 195.079,A -85,B 0,C 180,E1 -4128.702,E2 -4128.702} C_VEL
LIN {X 0,Y 538.082,Z 195.084,A -85,B 0,C 180,E1 -4131.74,E2 -4131.74} C_VEL
LIN {X 0,Y 538.158,Z 195.07,A -85,B 0,C 180,E1 -4134.755,E2 -4134.755} C_VEL
LIN {X 0,Y 538.157,Z 195.074,A -85,B 0,C 180,E1 -4137.755,E2 -4137.755} C_VEL
LIN {X 0,Y 538.177,Z 195.067,A -85,B 0,C 180,E1 -4140.748,E2 -4140.748} C_VEL
LIN {X 0,Y 538.134,Z 195.077,A -85,B 0,C 180,E1 -4142.995,E2 -4142.995} C_VEL
LIN {X 0,Y 538.116,Z 195.076,A -85,B 0,C 180,E1 -4145.997,E2 -4145.997} C_VEL
LIN {X 0,Y 538.069,Z 195.085,A -85,B 0,C 180,E1 -4149.018,E2 -4149.018} C_VEL
LIN {X 0,Y 538.075,Z 195.079,A -85,B 0,C 180,E1 -4152.063,E2 -4152.063} C_VEL
LIN {X 0,Y 538.037,Z 195.094,A -85,B 0,C 180,E1 -4155.144,E2 -4155.144} C_VEL
LIN {X 0,Y 538.026,Z 195.086,A -85,B 0,C 180,E1 -4158.27,E2 -4158.27} C_VEL
LIN {X 0,Y 538.031,Z 195.088,A -85,B 0,C 180,E1 -4160.652,E2 -4160.652} C_VEL
LIN {X 0,Y 538.016,Z 195.086,A -85,B 0,C 180,E1 -4163.888,E2 -4163.888} C_VEL
LIN {X 0,Y 538.035,Z 195.079,A -85,B 0,C 180,E1 -4166.367,E2 -4166.367} C_VEL
LIN {X 0,Y 538.049,Z 195.091,A -85,B 0,C 180,E1 -4168.939,E2 -4168.939} C_VEL
LIN {X 0,Y 538.02,Z 195.087,A -85,B 0,C 180,E1 -4171.891,E2 -4171.891} C_VEL
LIN {X 0,Y 538.025,Z 195.09,A -85,B 0,C 180,E1 -4174.622,E2 -4174.622} C_VEL
LIN {X 0,Y 538.002,Z 195.094,A -85,B 0,C 180,E1 -4177.171,E2 -4177.171} C_VEL
LIN {X 0,Y 538.017,Z 195.088,A -85,B 0,C 180,E1 -4180.274,E2 -4180.274} C_VEL
LIN {X 0,Y 537.367,Z 195.175,A -85,B 0,C 180,E1 -4180.899,E2 -4180.899} C_VEL
LIN {X 0,Y 534.516,Z 195.53,A -85,B 0,C 180,E1 -4181.914,E2 -4181.914} C_VEL
LIN {X 0,Y 532.092,Z 195.832,A -85,B 0,C 180,E1 -4182.731,E2 -4182.731} C_VEL
LIN {X 0,Y 531.044,Z 195.957,A -85,B 0,C 180,E1 -4183.362,E2 -4183.362} C_VEL
LIN {X 0,Y 530.957,Z 195.967,A -85,B 0,C 180,E1 -4183.576,E2 -4183.576} C_VEL
LIN {X 0,Y 530.963,Z 195.972,A -85,B 0,C 180,E1 -4186.506,E2 -4186.506} C_VEL
LIN {X 0,Y 530.985,Z 195.97,A -85,B 0,C 180,E1 -4188.977,E2 -4188.977} C_VEL
LIN {X 0,Y 530.954,Z 195.968,A -85,B 0,C 180,E1 -4191.53,E2 -4191.53} C_VEL
LIN {X 0,Y 530.952,Z 195.972,A -85,B 0,C 180,E1 -4194.381,E2 -4194.381} C_VEL
LIN {X 0,Y 530.969,Z 195.969,A -85,B 0,C 180,E1 -4197.134,E2 -4197.134} C_VEL
LIN {X 0,Y 530.968,Z 195.968,A -85,B 0,C 180,E1 -4199.804,E2 -4199.804} C_VEL
LIN {X 0,Y 531.014,Z 195.967,A -85,B 0,C 180,E1 -4202.468,E2 -4202.468} C_VEL
LIN {X 0,Y 531.032,Z 196.104,A -85,B 0,C 180,E1 -4205.44,E2 -4205.44} C_VEL
LIN {X 0,Y 532.885,Z 204.915,A -85,B 0,C 180,E1 -4206.899,E2 -4206.899} C_VEL
LIN {X 0,Y 532.567,Z 217.819,A -85,B 0,C 180,E1 -4208.845,E2 -4208.845} C_VEL
LIN {X 0,Y 535.182,Z 229.648,A -85,B 0,C 180,E1 -4209.128,E2 -4209.128} C_VEL
LIN {X 0,Y 534.506,Z 353.022,A -85,B 0,C 180,E1 -4210.832,E2 -4210.832} C_VEL
LIN {X 0,Y 534.288,Z 383.707,A -85,B 0,C 180,E1 -4211.278,E2 -4211.278} C_VEL
LIN {X 0,Y 534.035,Z 399.341,A -85,B 0,C 180,E1 -4211.663,E2 -4211.663} C_VEL
LIN {X 0,Y 533.711,Z 413.819,A -85,B 0,C 180,E1 -4212.172,E2 -4212.172} C_VEL
LIN {X 0,Y 533.385,Z 426.505,A -85,B 0,C 180,E1 -4212.755,E2 -4212.755} C_VEL
LIN {X 0,Y 532.941,Z 440.112,A -85,B 0,C 180,E1 -4213.53,E2 -4213.53} C_VEL
LIN {X 0,Y 532.456,Z 453.689,A -85,B 0,C 180,E1 -4214.481,E2 -4214.481} C_VEL
LIN {X 0,Y 532.061,Z 465.273,A -85,B 0,C 180,E1 -4215.465,E2 -4215.465} C_VEL
LIN {X 0,Y 531.651,Z 476.744,A -85,B 0,C 180,E1 -4216.625,E2 -4216.625} C_VEL
LIN {X 0,Y 531.306,Z 486.395,A -85,B 0,C 180,E1 -4217.782,E2 -4217.782} C_VEL
LIN {X 0,Y 531.05,Z 495.851,A -85,B 0,C 180,E1 -4219.13,E2 -4219.13} C_VEL
LIN {X 0,Y 530.788,Z 504.723,A -85,B 0,C 180,E1 -4220.666,E2 -4220.666} C_VEL
LIN {X 0,Y 530.641,Z 511.073,A -85,B 0,C 180,E1 -4222.006,E2 -4222.006} C_VEL
LIN {X 0,Y 530.544,Z 516.693,A -85,B 0,C 180,E1 -4223.469,E2 -4223.469} C_VEL
LIN {X 0,Y 530.508,Z 520.358,A -85,B 0,C 180,E1 -4224.679,E2 -4224.679} C_VEL
LIN {X 0,Y 530.481,Z 523.862,A -85,B 0,C 180,E1 -4226.202,E2 -4226.202} C_VEL
LIN {X 0,Y 530.409,Z 526.184,A -85,B 0,C 180,E1 -4227.722,E2 -4227.722} C_VEL
LIN {X 0,Y 530.34,Z 527.375,A -85,B 0,C 180,E1 -4229.241,E2 -4229.241} C_VEL
LIN {X 0,Y 530.341,Z 527.394,A -85,B 0,C 180,E1 -4230.759,E2 -4230.759} C_VEL
LIN {X 0,Y 530.41,Z 526.282,A -85,B 0,C 180,E1 -4232.278,E2 -4232.278} C_VEL
LIN {X 0,Y 530.481,Z 524.036,A -85,B 0,C 180,E1 -4233.798,E2 -4233.798} C_VEL
LIN {X 0,Y 530.506,Z 520.606,A -85,B 0,C 180,E1 -4235.321,E2 -4235.321} C_VEL
LIN {X 0,Y 530.55,Z 515.909,A -85,B 0,C 180,E1 -4236.847,E2 -4236.847} C_VEL
LIN {X 0,Y 530.666,Z 509.82,A -85,B 0,C 180,E1 -4238.377,E2 -4238.377} C_VEL
LIN {X 0,Y 530.836,Z 502.153,A -85,B 0,C 180,E1 -4239.91,E2 -4239.91} C_VEL
LIN {X 0,Y 531.062,Z 493.974,A -85,B 0,C 180,E1 -4241.256,E2 -4241.256} C_VEL
LIN {X 0,Y 531.373,Z 484.124,A -85,B 0,C 180,E1 -4242.605,E2 -4242.605} C_VEL
LIN {X 0,Y 531.742,Z 474.02,A -85,B 0,C 180,E1 -4243.763,E2 -4243.763} C_VEL
LIN {X 0,Y 532.126,Z 461.993,A -85,B 0,C 180,E1 -4244.924,E2 -4244.924} C_VEL
LIN {X 0,Y 532.612,Z 449.894,A -85,B 0,C 180,E1 -4245.893,E2 -4245.893} C_VEL
LIN {X 0,Y 533.061,Z 436.83,A -85,B 0,C 180,E1 -4246.762,E2 -4246.762} C_VEL
LIN {X 0,Y 533.442,Z 424.354,A -85,B 0,C 180,E1 -4247.441,E2 -4247.441} C_VEL
LIN {X 0,Y 533.802,Z 409.762,A -85,B 0,C 180,E1 -4248.072,E2 -4248.072} C_VEL
LIN {X 0,Y 534.101,Z 394.317,A -85,B 0,C 180,E1 -4248.567,E2 -4248.567} C_VEL
LIN {X 0,Y 534.362,Z 378.821,A -85,B 0,C 180,E1 -4248.895,E2 -4248.895} C_VEL
LIN {X 0,Y 535.226,Z 230.173,A -85,B 0,C 180,E1 -4250.952,E2 -4250.952} C_VEL
LIN {X 0,Y 532.595,Z 217.735,A -85,B 0,C 180,E1 -4251.256,E2 -4251.256} C_VEL
LIN {X 0,Y 532.935,Z 205.638,A -85,B 0,C 180,E1 -4253.078,E2 -4253.078} C_VEL
LIN {X 0,Y 531.01,Z 195.967,A -85,B 0,C 180,E1 -4254.691,E2 -4254.691} C_VEL
LIN {X 0,Y 531.015,Z 195.969,A -85,B 0,C 180,E1 -4257.595,E2 -4257.595} C_VEL
LIN {X 0,Y 530.973,Z 195.967,A -85,B 0,C 180,E1 -4260.644,E2 -4260.644} C_VEL
LIN {X 0,Y 530.988,Z 195.969,A -85,B 0,C 180,E1 -4263.772,E2 -4263.772} C_VEL
LIN {X 0,Y 530.963,Z 195.967,A -85,B 0,C 180,E1 -4266.557,E2 -4266.557} C_VEL
LIN {X 0,Y 530.98,Z 195.966,A -85,B 0,C 180,E1 -4269.854,E2 -4269.854} C_VEL
LIN {X 0,Y 530.979,Z 195.964,A -85,B 0,C 180,E1 -4272.455,E2 -4272.455} C_VEL
LIN {X 0,Y 530.983,Z 195.968,A -85,B 0,C 180,E1 -4275.62,E2 -4275.62} C_VEL
LIN {X 0,Y 531.002,Z 195.96,A -85,B 0,C 180,E1 -4278.565,E2 -4278.565} C_VEL
LIN {X 0,Y 530.953,Z 195.967,A -85,B 0,C 180,E1 -4281.529,E2 -4281.529} C_VEL
LIN {X 0,Y 530.976,Z 195.964,A -85,B 0,C 180,E1 -4284.381,E2 -4284.381} C_VEL
LIN {X 0,Y 530.965,Z 195.97,A -85,B 0,C 180,E1 -4287.133,E2 -4287.133} C_VEL
LIN {X 0,Y 530.979,Z 195.963,A -85,B 0,C 180,E1 -4289.804,E2 -4289.804} C_VEL
LIN {X 0,Y 531.008,Z 195.962,A -85,B 0,C 180,E1 -4292.466,E2 -4292.466} C_VEL
LIN {X 0,Y 530.997,Z 195.969,A -85,B 0,C 180,E1 -4294.942,E2 -4294.942} C_VEL
LIN {X 0,Y 530.963,Z 195.965,A -85,B 0,C 180,E1 -4298.246,E2 -4298.246} C_VEL
LIN {X 0,Y 530.989,Z 195.968,A -85,B 0,C 180,E1 -4300.677,E2 -4300.677} C_VEL
LIN {X 0,Y 530.985,Z 195.97,A -85,B 0,C 180,E1 -4303.071,E2 -4303.071} C_VEL
LIN {X 0,Y 531.01,Z 195.959,A -85,B 0,C 180,E1 -4305.436,E2 -4305.436} C_VEL
LIN {X 0,Y 531.037,Z 195.962,A -85,B 0,C 180,E1 -4308.55,E2 -4308.55} C_VEL
LIN {X 0,Y 531.048,Z 195.955,A -85,B 0,C 180,E1 -4311.629,E2 -4311.629} C_VEL
LIN {X 0,Y 531.115,Z 195.953,A -85,B 0,C 180,E1 -4314.685,E2 -4314.685} C_VEL
LIN {X 0,Y 531.129,Z 195.945,A -85,B 0,C 180,E1 -4317.725,E2 -4317.725} C_VEL
LIN {X 0,Y 531.147,Z 195.951,A -85,B 0,C 180,E1 -4320.758,E2 -4320.758} C_VEL
LIN {X 0,Y 531.101,Z 195.95,A -85,B 0,C 180,E1 -4323.034,E2 -4323.034} C_VEL
LIN {X 0,Y 531.074,Z 195.954,A -85,B 0,C 180,E1 -4326.077,E2 -4326.077} C_VEL
LIN {X 0,Y 531.027,Z 195.959,A -85,B 0,C 180,E1 -4329.138,E2 -4329.138} C_VEL
LIN {X 0,Y 531.032,Z 195.963,A -85,B 0,C 180,E1 -4332.225,E2 -4332.225} C_VEL
LIN {X 0,Y 530.987,Z 195.964,A -85,B 0,C 180,E1 -4335.35,E2 -4335.35} C_VEL
LIN {X 0,Y 531.007,Z 195.959,A -85,B 0,C 180,E1 -4337.723,E2 -4337.723} C_VEL
LIN {X 0,Y 530.993,Z 195.963,A -85,B 0,C 180,E1 -4340.938,E2 -4340.938} C_VEL
LIN {X 0,Y 530.971,Z 195.974,A -85,B 0,C 180,E1 -4344.225,E2 -4344.225} C_VEL
LIN {X 0,Y 530.998,Z 195.965,A -85,B 0,C 180,E1 -4346.744,E2 -4346.744} C_VEL
LIN {X 0,Y 530.992,Z 195.963,A -85,B 0,C 180,E1 -4349.322,E2 -4349.322} C_VEL
LIN {X 0,Y 530.973,Z 195.973,A -85,B 0,C 180,E1 -4352.104,E2 -4352.104} C_VEL
LIN {X 0,Y 530.981,Z 195.965,A -85,B 0,C 180,E1 -4354.855,E2 -4354.855} C_VEL
LIN {X 0,Y 530.959,Z 195.968,A -85,B 0,C 180,E1 -4357.508,E2 -4357.508} C_VEL
LIN {X 0,Y 530.978,Z 195.964,A -85,B 0,C 180,E1 -4360.433,E2 -4360.433} C_VEL
LIN {X 0,Y 530.96,Z 195.967,A -85,B 0,C 180,E1 -4363.282,E2 -4363.282} C_VEL
LIN {X 0,Y 530.981,Z 195.968,A -85,B 0,C 180,E1 -4365.622,E2 -4365.622} C_VEL
LIN {X 0,Y 531.003,Z 195.963,A -85,B 0,C 180,E1 -4368.566,E2 -4368.566} C_VEL
LIN {X 0,Y 530.964,Z 195.968,A -85,B 0,C 180,E1 -4371.347,E2 -4371.347} C_VEL
LIN {X 0,Y 530.973,Z 195.969,A -85,B 0,C 180,E1 -4374.382,E2 -4374.382} C_VEL
LIN {X 0,Y 530.967,Z 195.968,A -85,B 0,C 180,E1 -4377.134,E2 -4377.134} C_VEL
LIN {X 0,Y 530.967,Z 195.974,A -85,B 0,C 180,E1 -4379.804,E2 -4379.804} C_VEL
LIN {X 0,Y 531.019,Z 196.083,A -85,B 0,C 180,E1 -4382.261,E2 -4382.261} C_VEL
LIN {X 0,Y 533.607,Z 207.642,A -85,B 0,C 180,E1 -4383.947,E2 -4383.947} C_VEL
LIN {X 0,Y 533.121,Z 227.175,A -85,B 0,C 180,E1 -4386.499,E2 -4386.499} C_VEL
LIN {X 0,Y 532.61,Z 245.047,A -85,B 0,C 180,E1 -4388.795,E2 -4388.795} C_VEL
LIN {X 0,Y 535.081,Z 257.699,A -85,B 0,C 180,E1 -4389.076,E2 -4389.076} C_VEL
LIN {X 0,Y 534.465,Z 381.456,A -85,B 0,C 180,E1 -4390.783,E2 -4390.783} C_VEL
LIN {X 0,Y 534.242,Z 412.399,A -85,B 0,C 180,E1 -4391.233,E2 -4391.233} C_VEL
LIN {X 0,Y 533.977,Z 427.855,A -85,B 0,C 180,E1 -4391.611,E2 -4391.611} C_VEL
LIN {X 0,Y 533.631,Z 442.444,A -85,B 0,C 180,E1 -4392.12,E2 -4392.12} C_VEL
LIN {X 0,Y 533.201,Z 456.232,A -85,B 0,C 180,E1 -4392.749,E2 -4392.749} C_VEL
LIN {X 0,Y 532.803,Z 469.749,A -85,B 0,C 180,E1 -4393.525,E2 -4393.525} C_VEL
LIN {X 0,Y 532.408,Z 482.381,A -85,B 0,C 180,E1 -4394.411,E2 -4394.411} C_VEL
LIN {X 0,Y 531.943,Z 494.895,A -85,B 0,C 180,E1 -4395.462,E2 -4395.462} C_VEL
LIN {X 0,Y 531.566,Z 506.418,A -85,B 0,C 180,E1 -4396.622,E2 -4396.622} C_VEL
LIN {X 0,Y 531.254,Z 516.118,A -85,B 0,C 180,E1 -4397.78,E2 -4397.78} C_VEL
LIN {X 0,Y 531.033,Z 525.647,A -85,B 0,C 180,E1 -4399.13,E2 -4399.13} C_VEL
LIN {X 0,Y 530.739,Z 533.583,A -85,B 0,C 180,E1 -4400.473,E2 -4400.473} C_VEL
LIN {X 0,Y 530.613,Z 540.995,A -85,B 0,C 180,E1 -4402.006,E2 -4402.006} C_VEL
LIN {X 0,Y 530.545,Z 546.651,A -85,B 0,C 180,E1 -4403.467,E2 -4403.467} C_VEL
LIN {X 0,Y 530.509,Z 550.37,A -85,B 0,C 180,E1 -4404.679,E2 -4404.679} C_VEL
LIN {X 0,Y 530.48,Z 553.886,A -85,B 0,C 180,E1 -4406.202,E2 -4406.202} C_VEL
LIN {X 0,Y 530.409,Z 556.188,A -85,B 0,C 180,E1 -4407.722,E2 -4407.722} C_VEL
LIN {X 0,Y 530.342,Z 557.347,A -85,B 0,C 180,E1 -4409.241,E2 -4409.241} C_VEL
LIN {X 0,Y 530.342,Z 557.346,A -85,B 0,C 180,E1 -4410.759,E2 -4410.759} C_VEL
LIN {X 0,Y 530.409,Z 556.184,A -85,B 0,C 180,E1 -4412.278,E2 -4412.278} C_VEL
LIN {X 0,Y 530.48,Z 553.881,A -85,B 0,C 180,E1 -4413.798,E2 -4413.798} C_VEL
LIN {X 0,Y 530.509,Z 550.371,A -85,B 0,C 180,E1 -4415.321,E2 -4415.321} C_VEL
LIN {X 0,Y 530.569,Z 545.553,A -85,B 0,C 180,E1 -4416.847,E2 -4416.847} C_VEL
LIN {X 0,Y 530.665,Z 539.313,A -85,B 0,C 180,E1 -4418.377,E2 -4418.377} C_VEL
LIN {X 0,Y 530.808,Z 531.475,A -85,B 0,C 180,E1 -4419.911,E2 -4419.911} C_VEL
LIN {X 0,Y 531.029,Z 523.141,A -85,B 0,C 180,E1 -4421.257,E2 -4421.257} C_VEL
LIN {X 0,Y 531.328,Z 513.101,A -85,B 0,C 180,E1 -4422.606,E2 -4422.606} C_VEL
LIN {X 0,Y 531.688,Z 502.834,A -85,B 0,C 180,E1 -4423.764,E2 -4423.764} C_VEL
LIN {X 0,Y 532.105,Z 490.605,A -85,B 0,C 180,E1 -4424.925,E2 -4424.925} C_VEL
LIN {X 0,Y 532.521,Z 478.335,A -85,B 0,C 180,E1 -4425.893,E2 -4425.893} C_VEL
LIN {X 0,Y 533.005,Z 464.983,A -85,B 0,C 180,E1 -4426.764,E2 -4426.764} C_VEL
LIN {X 0,Y 533.386,Z 450.252,A -85,B 0,C 180,E1 -4427.542,E2 -4427.542} C_VEL
LIN {X 0,Y 533.809,Z 434.7,A -85,B 0,C 180,E1 -4428.171,E2 -4428.171} C_VEL
LIN {X 0,Y 534.126,Z 419.176,A -85,B 0,C 180,E1 -4428.623,E2 -4428.623} C_VEL
LIN {X 0,Y 534.329,Z 402.807,A -85,B 0,C 180,E1 -4428.925,E2 -4428.925} C_VEL
LIN {X 0,Y 535.173,Z 258.972,A -85,B 0,C 180,E1 -4430.902,E2 -4430.902} C_VEL
LIN {X 0,Y 532.62,Z 245.008,A -85,B 0,C 180,E1 -4431.21,E2 -4431.21} C_VEL
LIN {X 0,Y 533.179,Z 224.025,A -85,B 0,C 180,E1 -4433.911,E2 -4433.911} C_VEL
LIN {X 0,Y 533.6,Z 207.646,A -85,B 0,C 180,E1 -4436.053,E2 -4436.053} C_VEL
LIN {X 0,Y 530.997,Z 195.97,A -85,B 0,C 180,E1 -4437.788,E2 -4437.788} C_VEL
LIN {X 0,Y 530.971,Z 195.967,A -85,B 0,C 180,E1 -4440.644,E2 -4440.644} C_VEL
LIN {X 0,Y 530.986,Z 195.963,A -85,B 0,C 180,E1 -4443.772,E2 -4443.772} C_VEL
LIN {X 0,Y 530.962,Z 195.97,A -85,B 0,C 180,E1 -4446.557,E2 -4446.557} C_VEL
LIN {X 0,Y 531.002,Z 195.968,A -85,B 0,C 180,E1 -4449.857,E2 -4449.857} C_VEL
LIN {X 0,Y 530.975,Z 195.967,A -85,B 0,C 180,E1 -4452.456,E2 -4452.456} C_VEL
LIN {X 0,Y 530.982,Z 195.967,A -85,B 0,C 180,E1 -4455.62,E2 -4455.62} C_VEL
LIN {X 0,Y 531.001,Z 195.962,A -85,B 0,C 180,E1 -4458.565,E2 -4458.565} C_VEL
LIN {X 0,Y 530.962,Z 195.967,A -85,B 0,C 180,E1 -4461.345,E2 -4461.345} C_VEL
LIN {X 0,Y 530.975,Z 195.965,A -85,B 0,C 180,E1 -4464.382,E2 -4464.382} C_VEL
LIN {X 0,Y 530.965,Z 195.965,A -85,B 0,C 180,E1 -4467.133,E2 -4467.133} C_VEL
LIN {X 0,Y 530.979,Z 195.971,A -85,B 0,C 180,E1 -4469.804,E2 -4469.804} C_VEL
LIN {X 0,Y 531.008,Z 195.96,A -85,B 0,C 180,E1 -4472.466,E2 -4472.466} C_VEL
LIN {X 0,Y 530.997,Z 195.962,A -85,B 0,C 180,E1 -4474.942,E2 -4474.942} C_VEL
LIN {X 0,Y 530.963,Z 195.961,A -85,B 0,C 180,E1 -4478.246,E2 -4478.246} C_VEL
LIN {X 0,Y 530.988,Z 195.962,A -85,B 0,C 180,E1 -4480.677,E2 -4480.677} C_VEL
LIN {X 0,Y 530.984,Z 195.965,A -85,B 0,C 180,E1 -4483.071,E2 -4483.071} C_VEL
LIN {X 0,Y 531.01,Z 195.967,A -85,B 0,C 180,E1 -4485.436,E2 -4485.436} C_VEL
LIN {X 0,Y 531.037,Z 195.956,A -85,B 0,C 180,E1 -4488.55,E2 -4488.55} C_VEL
LIN {X 0,Y 531.051,Z 195.961,A -85,B 0,C 180,E1 -4491.629,E2 -4491.629} C_VEL
LIN {X 0,Y 531.116,Z 195.947,A -85,B 0,C 180,E1 -4494.685,E2 -4494.685} C_VEL
LIN {X 0,Y 531.13,Z 195.95,A -85,B 0,C 180,E1 -4497.725,E2 -4497.725} C_VEL
LIN {X 0,Y 531.147,Z 195.943,A -85,B 0,C 180,E1 -4500.758,E2 -4500.758} C_VEL
LIN {X 0,Y 531.1,Z 195.954,A -85,B 0,C 180,E1 -4503.034,E2 -4503.034} C_VEL
LIN {X 0,Y 531.075,Z 195.953,A -85,B 0,C 180,E1 -4506.077,E2 -4506.077} C_VEL
LIN {X 0,Y 531.028,Z 195.963,A -85,B 0,C 180,E1 -4509.138,E2 -4509.138} C_VEL
LIN {X 0,Y 531.032,Z 195.956,A -85,B 0,C 180,E1 -4512.225,E2 -4512.225} C_VEL
LIN {X 0,Y 530.987,Z 195.969,A -85,B 0,C 180,E1 -4515.35,E2 -4515.35} C_VEL
LIN {X 0,Y 531.008,Z 195.962,A -85,B 0,C 180,E1 -4517.723,E2 -4517.723} C_VEL
LIN {X 0,Y 530.991,Z 195.968,A -85,B 0,C 180,E1 -4520.938,E2 -4520.938} C_VEL
LIN {X 0,Y 530.972,Z 195.964,A -85,B 0,C 180,E1 -4524.225,E2 -4524.225} C_VEL
LIN {X 0,Y 530.999,Z 195.958,A -85,B 0,C 180,E1 -4526.744,E2 -4526.744} C_VEL
LIN {X 0,Y 530.993,Z 195.967,A -85,B 0,C 180,E1 -4529.322,E2 -4529.322} C_VEL
LIN {X 0,Y 530.973,Z 195.965,A -85,B 0,C 180,E1 -4532.104,E2 -4532.104} C_VEL
LIN {X 0,Y 530.983,Z 195.97,A -85,B 0,C 180,E1 -4534.855,E2 -4534.855} C_VEL
LIN {X 0,Y 530.961,Z 195.967,A -85,B 0,C 180,E1 -4537.508,E2 -4537.508} C_VEL
LIN {X 0,Y 530.98,Z 195.966,A -85,B 0,C 180,E1 -4540.433,E2 -4540.433} C_VEL
LIN {X 0,Y 530.962,Z 195.968,A -85,B 0,C 180,E1 -4543.282,E2 -4543.282} C_VEL
LIN {X 0,Y 530.957,Z 195.967,A -85,B 0,C 180,E1 -4543.576,E2 -4543.576} C_VEL
LIN {X 0,Y 530.285,Z 196.052,A -85,B 0,C 180,E1 -4544.209,E2 -4544.209} C_VEL
LIN {X 0,Y 527.439,Z 196.414,A -85,B 0,C 180,E1 -4545.238,E2 -4545.238} C_VEL
LIN {X 0,Y 525.037,Z 196.717,A -85,B 0,C 180,E1 -4546.067,E2 -4546.067} C_VEL
LIN {X 0,Y 524.004,Z 196.843,A -85,B 0,C 180,E1 -4546.706,E2 -4546.706} C_VEL
LIN {X 0,Y 523.919,Z 196.851,A -85,B 0,C 180,E1 -4546.923,E2 -4546.923} C_VEL
LIN {X 0,Y 523.945,Z 196.842,A -85,B 0,C 180,E1 -4549.921,E2 -4549.921} C_VEL
LIN {X 0,Y 523.904,Z 196.852,A -85,B 0,C 180,E1 -4552.869,E2 -4552.869} C_VEL
LIN {X 0,Y 523.931,Z 196.844,A -85,B 0,C 180,E1 -4555.711,E2 -4555.711} C_VEL
LIN {X 0,Y 523.922,Z 196.851,A -85,B 0,C 180,E1 -4558.457,E2 -4558.457} C_VEL
LIN {X 0,Y 523.938,Z 196.846,A -85,B 0,C 180,E1 -4561.126,E2 -4561.126} C_VEL
LIN {X 0,Y 523.984,Z 196.842,A -85,B 0,C 180,E1 -4563.981,E2 -4563.981} C_VEL
LIN {X 0,Y 523.977,Z 196.956,A -85,B 0,C 180,E1 -4565.193,E2 -4565.193} C_VEL
LIN {X 0,Y 526.01,Z 206.435,A -85,B 0,C 180,E1 -4566.788,E2 -4566.788} C_VEL
LIN {X 0,Y 525.78,Z 218.269,A -85,B 0,C 180,E1 -4568.568,E2 -4568.568} C_VEL
LIN {X 0,Y 528.591,Z 230.922,A -85,B 0,C 180,E1 -4568.87,E2 -4568.87} C_VEL
LIN {X 0,Y 527.647,Z 381.408,A -85,B 0,C 180,E1 -4570.986,E2 -4570.986} C_VEL
LIN {X 0,Y 527.437,Z 395.563,A -85,B 0,C 180,E1 -4571.309,E2 -4571.309} C_VEL
LIN {X 0,Y 527.102,Z 408.936,A -85,B 0,C 180,E1 -4571.74,E2 -4571.74} C_VEL
LIN {X 0,Y 526.655,Z 422.764,A -85,B 0,C 180,E1 -4572.327,E2 -4572.327} C_VEL
LIN {X 0,Y 526.295,Z 435.595,A -85,B 0,C 180,E1 -4573.016,E2 -4573.016} C_VEL
LIN {X 0,Y 525.82,Z 448.971,A -85,B 0,C 180,E1 -4573.899,E2 -4573.899} C_VEL
LIN {X 0,Y 525.323,Z 461.208,A -85,B 0,C 180,E1 -4574.878,E2 -4574.878} C_VEL
LIN {X 0,Y 524.841,Z 473.404,A -85,B 0,C 180,E1 -4576.053,E2 -4576.053} C_VEL
LIN {X 0,Y 524.462,Z 483.592,A -85,B 0,C 180,E1 -4577.226,E2 -4577.226} C_VEL
LIN {X 0,Y 524.088,Z 493.564,A -85,B 0,C 180,E1 -4578.592,E2 -4578.592} C_VEL
LIN {X 0,Y 523.826,Z 501.834,A -85,B 0,C 180,E1 -4579.956,E2 -4579.956} C_VEL
LIN {X 0,Y 523.614,Z 509.6,A -85,B 0,C 180,E1 -4581.51,E2 -4581.51} C_VEL
LIN {X 0,Y 523.483,Z 515.784,A -85,B 0,C 180,E1 -4583.06,E2 -4583.06} C_VEL
LIN {X 0,Y 523.445,Z 520.56,A -85,B 0,C 180,E1 -4584.607,E2 -4584.607} C_VEL
LIN {X 0,Y 523.402,Z 524.063,A -85,B 0,C 180,E1 -4586.15,E2 -4586.15} C_VEL
LIN {X 0,Y 523.333,Z 526.385,A -85,B 0,C 180,E1 -4587.691,E2 -4587.691} C_VEL
LIN {X 0,Y 523.246,Z 527.575,A -85,B 0,C 180,E1 -4589.23,E2 -4589.23} C_VEL
LIN {X 0,Y 523.247,Z 527.595,A -85,B 0,C 180,E1 -4590.77,E2 -4590.77} C_VEL
LIN {X 0,Y 523.333,Z 526.481,A -85,B 0,C 180,E1 -4592.309,E2 -4592.309} C_VEL
LIN {X 0,Y 523.402,Z 524.236,A -85,B 0,C 180,E1 -4593.849,E2 -4593.849} C_VEL
LIN {X 0,Y 523.442,Z 520.805,A -85,B 0,C 180,E1 -4595.393,E2 -4595.393} C_VEL
LIN {X 0,Y 523.482,Z 516.108,A -85,B 0,C 180,E1 -4596.94,E2 -4596.94} C_VEL
LIN {X 0,Y 523.612,Z 510.019,A -85,B 0,C 180,E1 -4598.49,E2 -4598.49} C_VEL
LIN {X 0,Y 523.815,Z 502.351,A -85,B 0,C 180,E1 -4600.045,E2 -4600.045} C_VEL
LIN {X 0,Y 524.059,Z 494.172,A -85,B 0,C 180,E1 -4601.409,E2 -4601.409} C_VEL
LIN {X 0,Y 524.407,Z 484.321,A -85,B 0,C 180,E1 -4602.775,E2 -4602.775} C_VEL
LIN {X 0,Y 524.799,Z 474.216,A -85,B 0,C 180,E1 -4603.948,E2 -4603.948} C_VEL
LIN {X 0,Y 525.249,Z 462.187,A -85,B 0,C 180,E1 -4605.124,E2 -4605.124} C_VEL
LIN {X 0,Y 525.804,Z 448.838,A -85,B 0,C 180,E1 -4606.201,E2 -4606.201} C_VEL
LIN {X 0,Y 526.325,Z 435.445,A -85,B 0,C 180,E1 -4607.083,E2 -4607.083} C_VEL
LIN {X 0,Y 526.752,Z 420.545,A -85,B 0,C 180,E1 -4607.87,E2 -4607.87} C_VEL
LIN {X 0,Y 527.146,Z 406.038,A -85,B 0,C 180,E1 -4608.459,E2 -4608.459} C_VEL
LIN {X 0,Y 527.49,Z 390.324,A -85,B 0,C 180,E1 -4608.921,E2 -4608.921} C_VEL
LIN {X 0,Y 527.69,Z 374.779,A -85,B 0,C 180,E1 -4609.212,E2 -4609.212} C_VEL
LIN {X 0,Y 528.522,Z 230.546,A -85,B 0,C 180,E1 -4611.228,E2 -4611.228} C_VEL
LIN {X 0,Y 525.743,Z 217.99,A -85,B 0,C 180,E1 -4611.535,E2 -4611.535} C_VEL
LIN {X 0,Y 526.071,Z 207.014,A -85,B 0,C 180,E1 -4613.209,E2 -4613.209} C_VEL
LIN {X 0,Y 523.99,Z 196.842,A -85,B 0,C 180,E1 -4614.938,E2 -4614.938} C_VEL
LIN {X 0,Y 523.969,Z 196.843,A -85,B 0,C 180,E1 -4617.998,E2 -4617.998} C_VEL
LIN {X 0,Y 523.943,Z 196.844,A -85,B 0,C 180,E1 -4620.854,E2 -4620.854} C_VEL
LIN {X 0,Y 523.959,Z 196.845,A -85,B 0,C 180,E1 -4623.734,E2 -4623.734} C_VEL
LIN {X 0,Y 523.916,Z 196.845,A -85,B 0,C 180,E1 -4626.403,E2 -4626.403} C_VEL
LIN {X 0,Y 523.92,Z 196.851,A -85,B 0,C 180,E1 -4629.084,E2 -4629.084} C_VEL
LIN {X 0,Y 523.954,Z 196.84,A -85,B 0,C 180,E1 -4632.118,E2 -4632.118} C_VEL
LIN {X 0,Y 523.951,Z 196.849,A -85,B 0,C 180,E1 -4635.308,E2 -4635.308} C_VEL
LIN {X 0,Y 523.967,Z 196.837,A -85,B 0,C 180,E1 -4638.687,E2 -4638.687} C_VEL
LIN {X 0,Y 523.915,Z 196.852,A -85,B 0,C 180,E1 -4641.079,E2 -4641.079} C_VEL
LIN {X 0,Y 523.922,Z 196.843,A -85,B 0,C 180,E1 -4643.827,E2 -4643.827} C_VEL
LIN {X 0,Y 523.936,Z 196.844,A -85,B 0,C 180,E1 -4646.635,E2 -4646.635} C_VEL
LIN {X 0,Y 523.957,Z 196.842,A -85,B 0,C 180,E1 -4649.356,E2 -4649.356} C_VEL
LIN {X 0,Y 523.971,Z 196.838,A -85,B 0,C 180,E1 -4652.28,E2 -4652.28} C_VEL
LIN {X 0,Y 523.944,Z 196.842,A -85,B 0,C 180,E1 -4654.581,E2 -4654.581} C_VEL
LIN {X 0,Y 523.908,Z 196.85,A -85,B 0,C 180,E1 -4657.106,E2 -4657.106} C_VEL
LIN {X 0,Y 523.97,Z 196.837,A -85,B 0,C 180,E1 -4659.865,E2 -4659.865} C_VEL
LIN {X 0,Y 523.962,Z 196.845,A -85,B 0,C 180,E1 -4662.837,E2 -4662.837} C_VEL
LIN {X 0,Y 523.967,Z 196.839,A -85,B 0,C 180,E1 -4665.235,E2 -4665.235} C_VEL
LIN {X 0,Y 524.002,Z 196.836,A -85,B 0,C 180,E1 -4668.394,E2 -4668.394} C_VEL
LIN {X 0,Y 523.996,Z 196.834,A -85,B 0,C 180,E1 -4671.516,E2 -4671.516} C_VEL
LIN {X 0,Y 524.076,Z 196.83,A -85,B 0,C 180,E1 -4674.614,E2 -4674.614} C_VEL
LIN {X 0,Y 524.101,Z 196.821,A -85,B 0,C 180,E1 -4677.694,E2 -4677.694} C_VEL
LIN {X 0,Y 524.117,Z 196.827,A -85,B 0,C 180,E1 -4680.768,E2 -4680.768} C_VEL
LIN {X 0,Y 524.067,Z 196.826,A -85,B 0,C 180,E1 -4683.075,E2 -4683.075} C_VEL
LIN {X 0,Y 524.036,Z 196.832,A -85,B 0,C 180,E1 -4686.159,E2 -4686.159} C_VEL
LIN {X 0,Y 523.995,Z 196.834,A -85,B 0,C 180,E1 -4689.262,E2 -4689.262} C_VEL
LIN {X 0,Y 523.998,Z 196.835,A -85,B 0,C 180,E1 -4691.743,E2 -4691.743} C_VEL
LIN {X 0,Y 523.984,Z 196.838,A -85,B 0,C 180,E1 -4695.053,E2 -4695.053} C_VEL
LIN {X 0,Y 523.955,Z 196.84,A -85,B 0,C 180,E1 -4697.969,E2 -4697.969} C_VEL
LIN {X 0,Y 523.963,Z 196.846,A -85,B 0,C 180,E1 -4700.41,E2 -4700.41} C_VEL
LIN {X 0,Y 523.908,Z 196.848,A -85,B 0,C 180,E1 -4702.894,E2 -4702.894} C_VEL
LIN {X 0,Y 523.944,Z 196.839,A -85,B 0,C 180,E1 -4705.419,E2 -4705.419} C_VEL
LIN {X 0,Y 523.962,Z 196.844,A -85,B 0,C 180,E1 -4707.999,E2 -4707.999} C_VEL
LIN {X 0,Y 523.945,Z 196.842,A -85,B 0,C 180,E1 -4710.857,E2 -4710.857} C_VEL
LIN {X 0,Y 523.954,Z 196.841,A -85,B 0,C 180,E1 -4713.735,E2 -4713.735} C_VEL
LIN {X 0,Y 523.916,Z 196.849,A -85,B 0,C 180,E1 -4716.405,E2 -4716.405} C_VEL
LIN {X 0,Y 523.915,Z 196.843,A -85,B 0,C 180,E1 -4719.085,E2 -4719.085} C_VEL
LIN {X 0,Y 523.95,Z 196.846,A -85,B 0,C 180,E1 -4722.119,E2 -4722.119} C_VEL
LIN {X 0,Y 523.95,Z 196.841,A -85,B 0,C 180,E1 -4725.309,E2 -4725.309} C_VEL
LIN {X 0,Y 523.968,Z 196.839,A -85,B 0,C 180,E1 -4728.688,E2 -4728.688} C_VEL
LIN {X 0,Y 523.92,Z 196.844,A -85,B 0,C 180,E1 -4731.08,E2 -4731.08} C_VEL
LIN {X 0,Y 523.92,Z 196.851,A -85,B 0,C 180,E1 -4733.828,E2 -4733.828} C_VEL
LIN {X 0,Y 523.939,Z 196.844,A -85,B 0,C 180,E1 -4736.636,E2 -4736.636} C_VEL
LIN {X 0,Y 523.953,Z 196.843,A -85,B 0,C 180,E1 -4739.356,E2 -4739.356} C_VEL
LIN {X 0,Y 523.98,Z 196.958,A -85,B 0,C 180,E1 -4742.002,E2 -4742.002} C_VEL
LIN {X 0,Y 526.805,Z 209.653,A -85,B 0,C 180,E1 -4743.881,E2 -4743.881} C_VEL
LIN {X 0,Y 526.189,Z 230.292,A -85,B 0,C 180,E1 -4746.609,E2 -4746.609} C_VEL
LIN {X 0,Y 525.777,Z 245.147,A -85,B 0,C 180,E1 -4748.512,E2 -4748.512} C_VEL
LIN {X 0,Y 528.509,Z 259.352,A -85,B 0,C 180,E1 -4748.83,E2 -4748.83} C_VEL
LIN {X 0,Y 527.555,Z 410.862,A -85,B 0,C 180,E1 -4750.958,E2 -4750.958} C_VEL
LIN {X 0,Y 527.238,Z 426.881,A -85,B 0,C 180,E1 -4751.343,E2 -4751.343} C_VEL
LIN {X 0,Y 526.868,Z 442.243,A -85,B 0,C 180,E1 -4751.883,E2 -4751.883} C_VEL
LIN {X 0,Y 526.378,Z 456.03,A -85,B 0,C 180,E1 -4752.518,E2 -4752.518} C_VEL
LIN {X 0,Y 525.966,Z 469.547,A -85,B 0,C 180,E1 -4753.305,E2 -4753.305} C_VEL
LIN {X 0,Y 525.496,Z 482.925,A -85,B 0,C 180,E1 -4754.258,E2 -4754.258} C_VEL
LIN {X 0,Y 524.952,Z 495.766,A -85,B 0,C 180,E1 -4755.363,E2 -4755.363} C_VEL
LIN {X 0,Y 524.519,Z 507.987,A -85,B 0,C 180,E1 -4756.637,E2 -4756.637} C_VEL
LIN {X 0,Y 524.136,Z 518.856,A -85,B 0,C 180,E1 -4758.005,E2 -4758.005} C_VEL
LIN {X 0,Y 523.904,Z 527.905,A -85,B 0,C 180,E1 -4759.371,E2 -4759.371} C_VEL
LIN {X 0,Y 523.653,Z 535.411,A -85,B 0,C 180,E1 -4760.732,E2 -4760.732} C_VEL
LIN {X 0,Y 523.509,Z 542.417,A -85,B 0,C 180,E1 -4762.285,E2 -4762.285} C_VEL
LIN {X 0,Y 523.441,Z 547.926,A -85,B 0,C 180,E1 -4763.834,E2 -4763.834} C_VEL
LIN {X 0,Y 523.322,Z 552.088,A -85,B 0,C 180,E1 -4765.378,E2 -4765.378} C_VEL
LIN {X 0,Y 523.358,Z 555.009,A -85,B 0,C 180,E1 -4766.921,E2 -4766.921} C_VEL
LIN {X 0,Y 523.272,Z 556.748,A -85,B 0,C 180,E1 -4768.461,E2 -4768.461} C_VEL
LIN {X 0,Y 523.243,Z 557.344,A -85,B 0,C 180,E1 -4770,E2 -4770} C_VEL
LIN {X 0,Y 523.272,Z 556.746,A -85,B 0,C 180,E1 -4771.539,E2 -4771.539} C_VEL
LIN {X 0,Y 523.358,Z 555.004,A -85,B 0,C 180,E1 -4773.079,E2 -4773.079} C_VEL
LIN {X 0,Y 523.322,Z 552.086,A -85,B 0,C 180,E1 -4774.622,E2 -4774.622} C_VEL
LIN {X 0,Y 523.451,Z 547.93,A -85,B 0,C 180,E1 -4776.166,E2 -4776.166} C_VEL
LIN {X 0,Y 523.509,Z 542.418,A -85,B 0,C 180,E1 -4777.715,E2 -4777.715} C_VEL
LIN {X 0,Y 523.653,Z 535.405,A -85,B 0,C 180,E1 -4779.268,E2 -4779.268} C_VEL
LIN {X 0,Y 523.932,Z 526.679,A -85,B 0,C 180,E1 -4780.824,E2 -4780.824} C_VEL
LIN {X 0,Y 524.177,Z 517.408,A -85,B 0,C 180,E1 -4782.191,E2 -4782.191} C_VEL
LIN {X 0,Y 524.519,Z 507.986,A -85,B 0,C 180,E1 -4783.363,E2 -4783.363} C_VEL
LIN {X 0,Y 524.97,Z 495.772,A -85,B 0,C 180,E1 -4784.636,E2 -4784.636} C_VEL
LIN {X 0,Y 525.434,Z 484.419,A -85,B 0,C 180,E1 -4785.625,E2 -4785.625} C_VEL
LIN {X 0,Y 525.875,Z 471.065,A -85,B 0,C 180,E1 -4786.598,E2 -4786.598} C_VEL
LIN {X 0,Y 526.37,Z 457.84,A -85,B 0,C 180,E1 -4787.382,E2 -4787.382} C_VEL
LIN {X 0,Y 526.821,Z 443.384,A -85,B 0,C 180,E1 -4788.069,E2 -4788.069} C_VEL
LIN {X 0,Y 527.2,Z 429.198,A -85,B 0,C 180,E1 -4788.583,E2 -4788.583} C_VEL
LIN {X 0,Y 527.474,Z 414.342,A -85,B 0,C 180,E1 -4788.97,E2 -4788.97} C_VEL
LIN {X 0,Y 527.651,Z 393.321,A -85,B 0,C 180,E1 -4789.304,E2 -4789.304} C_VEL
LIN {X 0,Y 528.543,Z 259.77,A -85,B 0,C 180,E1 -4791.163,E2 -4791.163} C_VEL
LIN {X 0,Y 525.729,Z 244.763,A -85,B 0,C 180,E1 -4791.506,E2 -4791.506} C_VEL
LIN {X 0,Y 526.33,Z 225.414,A -85,B 0,C 180,E1 -4794.032,E2 -4794.032} C_VEL
LIN {X 0,Y 526.814,Z 209.654,A -85,B 0,C 180,E1 -4796.118,E2 -4796.118} C_VEL
LIN {X 0,Y 523.977,Z 196.845,A -85,B 0,C 180,E1 -4798.025,E2 -4798.025} C_VEL
LIN {X 0,Y 523.942,Z 196.841,A -85,B 0,C 180,E1 -4800.854,E2 -4800.854} C_VEL
LIN {X 0,Y 523.957,Z 196.838,A -85,B 0,C 180,E1 -4803.734,E2 -4803.734} C_VEL
